	        // Check which specific status changed, prepare code, change state and write new status into the old one.
	        IF (#i_UDT_DimensionsCheckStatus.Specific.ParcelTooLongError <> #s_UDT_DimensionsCheckStatusOld.Specific.ParcelTooLongError AND NOT #sx_SendAllProcedure)
	            OR (#sx_SendAllProcedure AND #ii_ErrorNumber = 0)
	        THEN
	            #sdi_Code := "DB_MFC_ErrorCode".DimensionsCheck_v2.ParcelTooLongError;
	            #si_State := BOOL_TO_INT(#i_UDT_DimensionsCheckStatus.Specific.ParcelTooLongError);
	            #s_UDT_DimensionsCheckStatusOld.Specific.ParcelTooLongError := #i_UDT_DimensionsCheckStatus.Specific.ParcelTooLongError;
	            #sx_ItemErrorMessageReq := TRUE;
	            #ii_ErrorNumber += 1;
	        ELSIF (#i_UDT_DimensionsCheckStatus.Specific.ParcelTooShortError <> #s_UDT_DimensionsCheckStatusOld.Specific.ParcelTooShortError AND NOT #sx_SendAllProcedure)
	            OR (#sx_SendAllProcedure AND #ii_ErrorNumber = 1)
	        THEN
	            #sdi_Code := "DB_MFC_ErrorCode".DimensionsCheck_v2.ParcelTooShortError;
	            #si_State := BOOL_TO_INT(#i_UDT_DimensionsCheckStatus.Specific.ParcelTooShortError);
	            #s_UDT_DimensionsCheckStatusOld.Specific.ParcelTooShortError := #i_UDT_DimensionsCheckStatus.Specific.ParcelTooShortError;
	            #sx_ItemErrorMessageReq := TRUE;
	            #ii_ErrorNumber += 1;
	        ELSIF (#i_UDT_DimensionsCheckStatus.Specific.ParcelTooHighError <> #s_UDT_DimensionsCheckStatusOld.Specific.ParcelTooHighError AND NOT #sx_SendAllProcedure)
	            OR (#sx_SendAllProcedure AND #ii_ErrorNumber = 2)
	        THEN
	            #sdi_Code := "DB_MFC_ErrorCode".DimensionsCheck_v2.ParcelTooHighError;
	            #si_State := BOOL_TO_INT(#i_UDT_DimensionsCheckStatus.Specific.ParcelTooHighError);
	            #s_UDT_DimensionsCheckStatusOld.Specific.ParcelTooHighError := #i_UDT_DimensionsCheckStatus.Specific.ParcelTooHighError;
	            #sx_ItemErrorMessageReq := TRUE;
	            #ii_ErrorNumber += 1;
	        ELSIF (#i_UDT_DimensionsCheckStatus.Specific.ParcelTooLowError <> #s_UDT_DimensionsCheckStatusOld.Specific.ParcelTooLowError AND NOT #sx_SendAllProcedure)
	            OR (#sx_SendAllProcedure AND #ii_ErrorNumber = 3)
	        THEN
	            #sdi_Code := "DB_MFC_ErrorCode".DimensionsCheck_v2.ParcelTooLowError;
	            #si_State := BOOL_TO_INT(#i_UDT_DimensionsCheckStatus.Specific.ParcelTooLowError);
	            #s_UDT_DimensionsCheckStatusOld.Specific.ParcelTooLowError := #i_UDT_DimensionsCheckStatus.Specific.ParcelTooLowError;
	            #sx_ItemErrorMessageReq := TRUE;
	            #ii_ErrorNumber += 1;
	        ELSIF (#i_UDT_DimensionsCheckStatus.Specific.ParcelTooWideError <> #s_UDT_DimensionsCheckStatusOld.Specific.ParcelTooWideError AND NOT #sx_SendAllProcedure)
	            OR (#sx_SendAllProcedure AND #ii_ErrorNumber = 4)
	        THEN
	            #sdi_Code := "DB_MFC_ErrorCode".DimensionsCheck_v2.ParcelTooWideError;
	            #si_State := BOOL_TO_INT(#i_UDT_DimensionsCheckStatus.Specific.ParcelTooWideError);
	            #s_UDT_DimensionsCheckStatusOld.Specific.ParcelTooWideError := #i_UDT_DimensionsCheckStatus.Specific.ParcelTooWideError;
	            #sx_ItemErrorMessageReq := TRUE;
	            #ii_ErrorNumber += 1;
	        ELSIF (#i_UDT_DimensionsCheckStatus.Specific.ParcelTooNarrowError <> #s_UDT_DimensionsCheckStatusOld.Specific.ParcelTooNarrowError AND NOT #sx_SendAllProcedure)
	            OR (#sx_SendAllProcedure AND #ii_ErrorNumber = 5)
	        THEN
	            #sdi_Code := "DB_MFC_ErrorCode".DimensionsCheck_v2.ParcelTooNarrowError;
	            #si_State := BOOL_TO_INT(#i_UDT_DimensionsCheckStatus.Specific.ParcelTooNarrowError);
	            #s_UDT_DimensionsCheckStatusOld.Specific.ParcelTooNarrowError := #i_UDT_DimensionsCheckStatus.Specific.ParcelTooNarrowError;
	            #sx_ItemErrorMessageReq := TRUE;
	            #ii_ErrorNumber += 1;
	        ELSIF (#i_UDT_DimensionsCheckStatus.Specific.IncorrectParcelOrientationError <> #s_UDT_DimensionsCheckStatusOld.Specific.IncorrectParcelOrientationError AND NOT #sx_SendAllProcedure)
	            OR (#sx_SendAllProcedure AND #ii_ErrorNumber = 6)
	        THEN
	            #sdi_Code := "DB_MFC_ErrorCode".DimensionsCheck_v2.IncorrectParcelOrientationError;
	            #si_State := BOOL_TO_INT(#i_UDT_DimensionsCheckStatus.Specific.IncorrectParcelOrientationError);
	            #s_UDT_DimensionsCheckStatusOld.Specific.IncorrectParcelOrientationError := #i_UDT_DimensionsCheckStatus.Specific.IncorrectParcelOrientationError;
	            #sx_ItemErrorMessageReq := TRUE;
	            #ii_ErrorNumber += 1;
	        ELSIF (#i_UDT_DimensionsCheckStatus.Specific.GeneralError <> #s_UDT_DimensionsCheckStatusOld.Specific.GeneralError AND NOT #sx_SendAllProcedure)
	            OR (#sx_SendAllProcedure AND #ii_ErrorNumber = 7)
	        THEN
	            #sdi_Code := "DB_MFC_ErrorCode".DimensionsCheck_v2.GeneralError;
	            #si_State := BOOL_TO_INT(#i_UDT_DimensionsCheckStatus.Specific.GeneralError);
	            #s_UDT_DimensionsCheckStatusOld.Specific.GeneralError := #i_UDT_DimensionsCheckStatus.Specific.GeneralError;
	            #sx_ItemErrorMessageReq := TRUE;
	            #ii_ErrorNumber += 1;
	        ELSIF (#i_UDT_DimensionsCheckStatus.Specific.DisabledGeneralFunctionality <> #s_UDT_DimensionsCheckStatusOld.Specific.DisabledGeneralFunctionality AND NOT #sx_SendAllProcedure)
	            OR (#sx_SendAllProcedure AND #ii_ErrorNumber = 8)
	        THEN
	            #sdi_Code := "DB_MFC_ErrorCode".DimensionsCheck_v2.DisabledGeneralFunctionality;
	            #si_State := BOOL_TO_INT(#i_UDT_DimensionsCheckStatus.Specific.DisabledGeneralFunctionality);
	            #s_UDT_DimensionsCheckStatusOld.Specific.DisabledGeneralFunctionality := #i_UDT_DimensionsCheckStatus.Specific.DisabledGeneralFunctionality;
	            #sx_ItemErrorMessageReq := TRUE;
	            #ii_ErrorNumber += 1;
	        ELSIF (#i_UDT_DimensionsCheckStatus.Specific.DisabledTooLongParcel <> #s_UDT_DimensionsCheckStatusOld.Specific.DisabledTooLongParcel AND NOT #sx_SendAllProcedure)
	            OR (#sx_SendAllProcedure AND #ii_ErrorNumber = 9)
	        THEN
	            #sdi_Code := "DB_MFC_ErrorCode".DimensionsCheck_v2.DisabledTooLongParcel;
	            #si_State := BOOL_TO_INT(#i_UDT_DimensionsCheckStatus.Specific.DisabledTooLongParcel);
	            #s_UDT_DimensionsCheckStatusOld.Specific.DisabledTooLongParcel := #i_UDT_DimensionsCheckStatus.Specific.DisabledTooLongParcel;
	            #sx_ItemErrorMessageReq := TRUE;
	            #ii_ErrorNumber += 1;
	        ELSIF (#i_UDT_DimensionsCheckStatus.Specific.DisabledTooShortParcelError <> #s_UDT_DimensionsCheckStatusOld.Specific.DisabledTooShortParcelError AND NOT #sx_SendAllProcedure)
	            OR (#sx_SendAllProcedure AND #ii_ErrorNumber = 10)
	        THEN
	            #sdi_Code := "DB_MFC_ErrorCode".DimensionsCheck_v2.DisabledTooShortParcelError;
	            #si_State := BOOL_TO_INT(#i_UDT_DimensionsCheckStatus.Specific.DisabledTooShortParcelError);
	            #s_UDT_DimensionsCheckStatusOld.Specific.DisabledTooShortParcelError := #i_UDT_DimensionsCheckStatus.Specific.DisabledTooShortParcelError;
	            #sx_ItemErrorMessageReq := TRUE;
	            #ii_ErrorNumber += 1;
	        ELSIF (#i_UDT_DimensionsCheckStatus.Specific.DisabledTooHighParcelError <> #s_UDT_DimensionsCheckStatusOld.Specific.DisabledTooHighParcelError AND NOT #sx_SendAllProcedure)
	            OR (#sx_SendAllProcedure AND #ii_ErrorNumber = 11)
	        THEN
	            #sdi_Code := "DB_MFC_ErrorCode".DimensionsCheck_v2.DisabledTooHighParcelError;
	            #si_State := BOOL_TO_INT(#i_UDT_DimensionsCheckStatus.Specific.DisabledTooHighParcelError);
	            #s_UDT_DimensionsCheckStatusOld.Specific.DisabledTooHighParcelError := #i_UDT_DimensionsCheckStatus.Specific.DisabledTooHighParcelError;
	            #sx_ItemErrorMessageReq := TRUE;
	            #ii_ErrorNumber += 1;
	        ELSIF (#i_UDT_DimensionsCheckStatus.Specific.DisabledTooLowParcelError <> #s_UDT_DimensionsCheckStatusOld.Specific.DisabledTooLowParcelError AND NOT #sx_SendAllProcedure)
	            OR (#sx_SendAllProcedure AND #ii_ErrorNumber = 12)
	        THEN
	            #sdi_Code := "DB_MFC_ErrorCode".DimensionsCheck_v2.DisabledTooLowParcelError;
	            #si_State := BOOL_TO_INT(#i_UDT_DimensionsCheckStatus.Specific.DisabledTooLowParcelError);
	            #s_UDT_DimensionsCheckStatusOld.Specific.DisabledTooLowParcelError := #i_UDT_DimensionsCheckStatus.Specific.DisabledTooLowParcelError;
	            #sx_ItemErrorMessageReq := TRUE;
	            #ii_ErrorNumber += 1;
	        ELSIF (#i_UDT_DimensionsCheckStatus.Specific.DisabledTooWideParcelError <> #s_UDT_DimensionsCheckStatusOld.Specific.DisabledTooWideParcelError AND NOT #sx_SendAllProcedure)
	            OR (#sx_SendAllProcedure AND #ii_ErrorNumber = 13)
	        THEN
	            #sdi_Code := "DB_MFC_ErrorCode".DimensionsCheck_v2.DisabledTooWideParcelError;
	            #si_State := BOOL_TO_INT(#i_UDT_DimensionsCheckStatus.Specific.DisabledTooWideParcelError);
	            #s_UDT_DimensionsCheckStatusOld.Specific.DisabledTooWideParcelError := #i_UDT_DimensionsCheckStatus.Specific.DisabledTooWideParcelError;
	            #sx_ItemErrorMessageReq := TRUE;
	            #ii_ErrorNumber += 1;
	        ELSIF (#i_UDT_DimensionsCheckStatus.Specific.DisabledTooNarrowParcelError <> #s_UDT_DimensionsCheckStatusOld.Specific.DisabledTooNarrowParcelError AND NOT #sx_SendAllProcedure)
	            OR (#sx_SendAllProcedure AND #ii_ErrorNumber = 14)
	        THEN
	            #sdi_Code := "DB_MFC_ErrorCode".DimensionsCheck_v2.DisabledTooNarrowParcelError;
	            #si_State := BOOL_TO_INT(#i_UDT_DimensionsCheckStatus.Specific.DisabledTooNarrowParcelError);
	            #s_UDT_DimensionsCheckStatusOld.Specific.DisabledTooNarrowParcelError := #i_UDT_DimensionsCheckStatus.Specific.DisabledTooNarrowParcelError;
	            #sx_ItemErrorMessageReq := TRUE;
	            #ii_ErrorNumber += 1;
	        ELSIF (#i_UDT_DimensionsCheckStatus.Specific.DisabledParcelOrientationError <> #s_UDT_DimensionsCheckStatusOld.Specific.DisabledParcelOrientationError AND NOT #sx_SendAllProcedure)
	            OR (#sx_SendAllProcedure AND #ii_ErrorNumber = 15)
	        THEN
	            #sdi_Code := "DB_MFC_ErrorCode".DimensionsCheck_v2.DisabledParcelOrientationError;
	            #si_State := BOOL_TO_INT(#i_UDT_DimensionsCheckStatus.Specific.DisabledParcelOrientationError);
	            #s_UDT_DimensionsCheckStatusOld.Specific.DisabledParcelOrientationError := #i_UDT_DimensionsCheckStatus.Specific.DisabledParcelOrientationError;
	            #sx_ItemErrorMessageReq := TRUE;
	            #sx_SendAllProcedure := FALSE;
	            #ii_ErrorNumber += 1;
	        END_IF;
	    END_IF;
	END_REGION

	REGION 4 - Write message components to the item error structure

	    #s_UDT_ItemError.ItemNumber := #i_UDT_EquipmentNumber;
	    #s_UDT_ItemError.Error := #sdi_Code;
	    #s_UDT_ItemError.State := #si_State;
	    #s_UDT_ItemError.Masked := 1;

	END_REGION

	REGION 5 - Write message components to the item status structure

	    #s_UDT_ItemStatus.Group := #i_UDT_EquipmentNumber.Group;
	    #s_UDT_ItemStatus.Node := #i_UDT_EquipmentNumber.Node;
	    #s_UDT_ItemStatus.Status := #si_ItemStatus;

	END_REGION

	REGION 6 - Prepare messages to the MFC

	    // If item error message required signal is set, prepare the item error message.
	    IF (#sx_ItemErrorMessageReq)
	    THEN
	        #s_FB_ItemError(i_UDT_ItemErrorBody := #s_UDT_ItemError,
	                        ii_MessageGroup := 1,
	                        ix_FlagRetry := FALSE,
	                        idi_TimeSpan := 0,
	                        qx_Error => #sx_ItemErrorBlockError,
	                        qx_Warning => #sx_ItemErrorBlockWarning,
	                        iq_UDT_FifoHeader := #iq_UDT_FifoHeader,
	                        iqs_FifoData := #iqs_FifoData,
	                        iqdi_MessageSequenceNumber := #iqdi_MessageSequenceNumber);
	    END_IF;

	    // If item status message required signal is set, prepare the item error message.
	    IF (#sx_ItemStatusMessageReq)
	    THEN
	        #s_FB_ItemStatus(i_UDT_ItemStatusBody := #s_UDT_ItemStatus,
	                         ii_MessageGroup := 1,
	                         ix_FlagRetry := FALSE,
	                         idi_TimeSpan := 0,
	                         qx_Error => #sx_ItemStatusBlockError,
	                         qx_Warning => #sx_ItemStatusBlockWarning,
	                         iq_UDT_FifoHeader := #iq_UDT_FifoHeader,
	                         iqs_FifoData := #iqs_FifoData,
	                         iqdi_MessageSequenceNumber := #iqdi_MessageSequenceNumber);
	    END_IF;

	END_REGION

	REGION 7 - Write outputs

	    // Prepare collective output error.
	    #qx_Error :=
	    #sx_ItemErrorBlockError
	    OR #sx_ItemStatusBlockError
	    OR #sx_FIFOError;

	    // Prepare collective output warning.
	    #qx_Warning :=
	    #sx_ItemErrorBlockWarning
	    OR #sx_ItemStatusBlockWarning
	    OR #sx_FIFOWarning;

	END_REGION




END_FUNCTION_BLOCK

FUNCTION_BLOCK "FB_MFC_Visu_RetractableRoller_Status"
{ S7_Optimized_Access := 'TRUE' }
VERSION : 0.1
// ATTRIBUTES
// AUTO_NUMBER = True
// BLOCK_NUMBER = 157
// END_ATTRIBUTES
   VAR_INPUT
      i_UDT_RetractrableRollerStatus { ExternalAccessible := 'False'; ExternalVisible := 'False'; ExternalWritable := 'False'} : "UDT_RetractrableRoller_Status";   // RetractrableRoller status structure
      i_UDT_EquipmentNumber { ExternalAccessible := 'False'; ExternalVisible := 'False'; ExternalWritable := 'False'} : "UDT_EquipmentNumber";   // Item number
      ix_SendAllErrorsState { ExternalAccessible := 'False'; ExternalVisible := 'False'; ExternalWritable := 'False'} : Bool;   // True - update all the messages
      ix_MFCConnected { ExternalAccessible := 'False'; ExternalVisible := 'False'; ExternalWritable := 'False'} : Bool;   // True - A connection to the MFC has been established
      ix_CollectiveReset { ExternalAccessible := 'False'; ExternalVisible := 'False'; ExternalWritable := 'False'} : Bool;   // True - Collective reset command of all system controls
   END_VAR

   VAR_OUTPUT
      qx_Error { ExternalAccessible := 'False'; ExternalVisible := 'False'; ExternalWritable := 'False'} : Bool;   // Block error
      qx_Warning { ExternalAccessible := 'False'; ExternalVisible := 'False'; ExternalWritable := 'False'} : Bool;   // Block warning
   END_VAR

   VAR_IN_OUT
      iq_UDT_FifoHeader : "UDT_FifoHeader";   // FIFO header
      iqs_FifoData : Array[*] of "UDT_MessageV2";   // FIFO data buffer
      iqdi_MessageSequenceNumber { ExternalAccessible := 'False'; ExternalVisible := 'False'; ExternalWritable := 'False'} : DInt;   // Message number
   END_VAR

   VAR
      s_FB_ItemError { ExternalAccessible := 'False'; ExternalVisible := 'False'; ExternalWritable := 'False'; S7_SetPoint := 'False'} : "FB_ItemError";   // Item error block's instance
      s_FB_ItemStatus { ExternalAccessible := 'False'; ExternalVisible := 'False'; ExternalWritable := 'False'; S7_SetPoint := 'False'} : "FB_ItemStatus";   // Item status block's instance
      ss_FIFOStatus { ExternalAccessible := 'False'; ExternalVisible := 'False'; ExternalWritable := 'False'; S7_SetPoint := 'False'} : "UDT_FifoStatus";   // Status structure
      s_UDT_Message { ExternalAccessible := 'False'; ExternalVisible := 'False'; ExternalWritable := 'False'; S7_SetPoint := 'False'} : "UDT_MessageV2";   // Message
      s_UDT_RetractrableRollerOld { ExternalAccessible := 'False'; ExternalVisible := 'False'; ExternalWritable := 'False'; S7_SetPoint := 'False'} : "UDT_RetractrableRoller_Status";   // RetractrableRoller status structure
      s_UDT_ItemError { ExternalAccessible := 'False'; ExternalVisible := 'False'; ExternalWritable := 'False'; S7_SetPoint := 'False'} : "UDT_ItemError";   // Item error message body structure
      s_UDT_ItemStatus { ExternalAccessible := 'False'; ExternalVisible := 'False'; ExternalWritable := 'False'; S7_SetPoint := 'False'} : "UDT_ItemStatus";   // Item status message body structure
      s_R_TRIG_Connection {InstructionName := 'R_TRIG'; LibVersion := '1.0'; ExternalAccessible := 'False'; ExternalVisible := 'False'; ExternalWritable := 'False'; S7_SetPoint := 'False'} : R_TRIG;   // Rising edge trigger connection reastablished
      s_F_TRIG_SendAllErrors {InstructionName := 'F_TRIG'; LibVersion := '1.0'; ExternalAccessible := 'False'; ExternalVisible := 'False'; ExternalWritable := 'False'; S7_SetPoint := 'False'} : F_TRIG;   // Falling edge trigger from signal send all errors
      sdi_Code { ExternalAccessible := 'False'; ExternalVisible := 'False'; ExternalWritable := 'False'} : DInt;   // Error code
      si_ItemStatus { ExternalAccessible := 'False'; ExternalVisible := 'False'; ExternalWritable := 'False'} : Int;   // Item status
      ii_ErrorNumber { ExternalAccessible := 'False'; ExternalVisible := 'False'; ExternalWritable := 'False'} : Int;   // Counter Error Number
      si_State { ExternalAccessible := 'False'; ExternalVisible := 'False'; ExternalWritable := 'False'} : Int;   // Error state
      sx_ItemErrorMessageReq { ExternalAccessible := 'False'; ExternalVisible := 'False'; ExternalWritable := 'False'} : Bool;   // Item error message required
      sx_ItemStatusMessageReq { ExternalAccessible := 'False'; ExternalVisible := 'False'; ExternalWritable := 'False'} : Bool;   // Item status message required
      sx_SendAllProcedure { ExternalAccessible := 'False'; ExternalVisible := 'False'; ExternalWritable := 'False'} : Bool;   // Send all procedure
      sx_FIFOError { ExternalAccessible := 'False'; ExternalVisible := 'False'; ExternalWritable := 'False'} : Bool;   // FIFO error
      sx_FIFOWarning { ExternalAccessible := 'False'; ExternalVisible := 'False'; ExternalWritable := 'False'} : Bool;   // FIFO warning
      sx_ItemErrorBlockError { ExternalAccessible := 'False'; ExternalVisible := 'False'; ExternalWritable := 'False'} : Bool;   // Item error block error
      sx_ItemErrorBlockWarning { ExternalAccessible := 'False'; ExternalVisible := 'False'; ExternalWritable := 'False'} : Bool;   // Item error block warning
      sx_ItemStatusBlockError { ExternalAccessible := 'False'; ExternalVisible := 'False'; ExternalWritable := 'False'} : Bool;   // Item status block error
      sx_ItemStatusBlockWarning { ExternalAccessible := 'False'; ExternalVisible := 'False'; ExternalWritable := 'False'} : Bool;   // Item status block warning
   END_VAR


BEGIN
	(*
	----------------------------------------------------------------------------------------
	|                                                                                      |
	|  Copyright  2023             FORTNA Europe BV                                        |
	|  All Rights Reserved         Netherlands                                             |
	|                                                                                      |
	----------------------------------------------------------------------------------------
	Version history:
	Date        | Version   | Author       | Remark
	----------------------------------------------------------------------------------------
	09/05/2023  | 1.0       | M. Diebel   | Release TIA 17 | DHL Munich 2023
	13/03/2023  | 1.1       | S. Nieswiec | Updated for new Baseline
	*)


	REGION 1 - Initialize message required signals

	    #sx_ItemErrorMessageReq := FALSE;
	    #sx_ItemStatusMessageReq := FALSE;

	    // On connection reestablish send last remembered status and error state ( status only when it's diffrent then 0 )
	    #s_R_TRIG_Connection(CLK := #ix_MFCConnected);

	    IF #s_R_TRIG_Connection.Q AND #si_ItemStatus <> 0
	    THEN
	        #sx_ItemStatusMessageReq := TRUE;
	    END_IF;

	    IF #s_R_TRIG_Connection.Q
	    THEN
	        #sx_ItemErrorMessageReq := TRUE;
	    END_IF;

	    // Prepare trigger on the collective reset signal.
	    #s_F_TRIG_SendAllErrors(CLK := #ix_SendAllErrorsState);

	    // When collective reset will go down, start send every equipment errors.
	    IF #s_F_TRIG_SendAllErrors.Q AND NOT #sx_SendAllProcedure
	    THEN
	        #ii_ErrorNumber := 0;
	        #sx_SendAllProcedure := TRUE;
	    END_IF;

	END_REGION

	REGION 2 - FIFO header status update

	    // Mode 'S' - FIFO register status update.
	    "FC_Fifo"(ic_Mode := 'S',
	              qUDT_Status => #ss_FIFOStatus,
	              qx_Error => #sx_FIFOError,
	              qx_Warning => #sx_FIFOWarning,
	              iqv_Data := #s_UDT_Message,
	              iqUDT_FifoHeader := #iq_UDT_FifoHeader,
	              iqv_DataBuffer := #iqs_FifoData);

	END_REGION

	REGION 3 - Prepare message data

	    // When there is no reset errors command, update status and errors.
	    IF NOT #ix_CollectiveReset
	        AND NOT #ss_FIFOStatus.FifoPreFull
	    THEN
	        // Status
	        IF (#i_UDT_RetractrableRollerStatus.Status <> #s_UDT_RetractrableRollerOld.Status OR (#sx_SendAllProcedure AND #ii_ErrorNumber = 0))
	        THEN
	            #sx_ItemStatusMessageReq := TRUE;
	            #si_ItemStatus := #i_UDT_RetractrableRollerStatus.Status;
	            #s_UDT_RetractrableRollerOld.Status := #i_UDT_RetractrableRollerStatus.Status;
	        END_IF;


	        // Check which specific status changed, prepare code, change state and write new status into the old one.
	        IF (#i_UDT_RetractrableRollerStatus.Specific.NoHomePosition <> #s_UDT_RetractrableRollerOld.Specific.NoHomePosition AND NOT #sx_SendAllProcedure)
	            OR (#sx_SendAllProcedure AND #ii_ErrorNumber = 0)
	        THEN
	            #sdi_Code := "DB_MFC_ErrorCode".Retractable.NoHomePosition;
	            #si_State := BOOL_TO_INT(#i_UDT_RetractrableRollerStatus.Specific.NoHomePosition);
	            #s_UDT_RetractrableRollerOld.Specific.NoHomePosition := #i_UDT_RetractrableRollerStatus.Specific.NoHomePosition;
	            #sx_ItemErrorMessageReq := TRUE;
	            #ii_ErrorNumber += 1;
	        ELSIF (#i_UDT_RetractrableRollerStatus.Specific.RollerError <> #s_UDT_RetractrableRollerOld.Specific.RollerError AND NOT #sx_SendAllProcedure)
	            OR (#sx_SendAllProcedure AND #ii_ErrorNumber = 1)
	        THEN
	            #sdi_Code := "DB_MFC_ErrorCode".Retractable.Errorr;
	            #si_State := BOOL_TO_INT(#i_UDT_RetractrableRollerStatus.Specific.RollerError);
	            #s_UDT_RetractrableRollerOld.Specific.RollerError := #i_UDT_RetractrableRollerStatus.Specific.RollerError;
	            #sx_ItemErrorMessageReq := TRUE;
	            #sx_SendAllProcedure := FALSE;
	        END_IF;
	    END_IF;
	END_REGION

	REGION 4 - Write message components to the item error structure

	    #s_UDT_ItemError.ItemNumber := #i_UDT_EquipmentNumber;
	    #s_UDT_ItemError.Error := #sdi_Code;
	    #s_UDT_ItemError.State := #si_State;
	    #s_UDT_ItemError.Masked := 1;

	END_REGION

	REGION 5 - Write message components to the item status structure

	    #s_UDT_ItemStatus.Group := #i_UDT_EquipmentNumber.Group;
	    #s_UDT_ItemStatus.Node := #i_UDT_EquipmentNumber.Node;
	    #s_UDT_ItemStatus.Status := #si_ItemStatus;

	END_REGION

	REGION 6 - Prepare messages to the MFC

	    // If item error message required signal is set, prepare the item error message.
	    IF (#sx_ItemErrorMessageReq)
	    THEN
	        #s_FB_ItemError(i_UDT_ItemErrorBody := #s_UDT_ItemError,
	                        ii_MessageGroup := 1,
	                        ix_FlagRetry := FALSE,
	                        idi_TimeSpan := 0,
	                        qx_Error => #sx_ItemErrorBlockError,
	                        qx_Warning => #sx_ItemErrorBlockWarning,
	                        iq_UDT_FifoHeader := #iq_UDT_FifoHeader,
	                        iqs_FifoData := #iqs_FifoData,
	                        iqdi_MessageSequenceNumber := #iqdi_MessageSequenceNumber);
	    END_IF;

	    // If item status message required signal is set, prepare the item error message.
	    IF (#sx_ItemStatusMessageReq)
	    THEN
	        #s_FB_ItemStatus(i_UDT_ItemStatusBody := #s_UDT_ItemStatus,
	                         ii_MessageGroup := 1,
	                         ix_FlagRetry := FALSE,
	                         idi_TimeSpan := 0,
	                         qx_Error => #sx_ItemStatusBlockError,
	                         qx_Warning => #sx_ItemStatusBlockWarning,
	                         iq_UDT_FifoHeader := #iq_UDT_FifoHeader,
	                         iqs_FifoData := #iqs_FifoData,
	                         iqdi_MessageSequenceNumber := #iqdi_MessageSequenceNumber);
	    END_IF;

	END_REGION

	REGION 7 - Write outputs

	    // Prepare collective output error.
	    #qx_Error :=
	    #sx_ItemErrorBlockError
	    OR #sx_ItemStatusBlockError
	    OR #sx_FIFOError;

	    // Prepare collective output warning.
	    #qx_Warning :=
	    #sx_ItemErrorBlockWarning
	    OR #sx_ItemStatusBlockWarning
	    OR #sx_FIFOWarning;

	END_REGION


END_FUNCTION_BLOCK

FUNCTION_BLOCK "FB_MFC_Visu_RIO_Status"
{ S7_Optimized_Access := 'TRUE' }
VERSION : 0.1
// ATTRIBUTES
// AUTO_NUMBER = True
// BLOCK_NUMBER = 158
// END_ATTRIBUTES
   VAR_INPUT
      i_UDT_RIOStatus { ExternalAccessible := 'False'; ExternalVisible := 'False'; ExternalWritable := 'False'} : "UDT_RIOStatus";   // RIO status structure
      i_UDT_EquipmentNumber { ExternalAccessible := 'False'; ExternalVisible := 'False'; ExternalWritable := 'False'} : "UDT_EquipmentNumber";   // Item number
      ix_SendAllErrorsState { ExternalAccessible := 'False'; ExternalVisible := 'False'; ExternalWritable := 'False'} : Bool;   // True - update all the messages
      ix_MFCConnected { ExternalAccessible := 'False'; ExternalVisible := 'False'; ExternalWritable := 'False'} : Bool;   // True - A connection to the MFC has been established
      ix_CollectiveReset { ExternalAccessible := 'False'; ExternalVisible := 'False'; ExternalWritable := 'False'} : Bool;   // True - Collective reset command of all system controls
   END_VAR

   VAR_OUTPUT
      qx_Error { ExternalAccessible := 'False'; ExternalVisible := 'False'; ExternalWritable := 'False'} : Bool;   // Block error
      qx_Warning { ExternalAccessible := 'False'; ExternalVisible := 'False'; ExternalWritable := 'False'} : Bool;   // Block warning
   END_VAR

   VAR_IN_OUT
      iq_UDT_FifoHeader : "UDT_FifoHeader";   // FIFO header
      iqs_FifoData : Array[*] of "UDT_MessageV2";   // FIFO data buffer
      iqdi_MessageSequenceNumber { ExternalAccessible := 'False'; ExternalVisible := 'False'; ExternalWritable := 'False'} : DInt;   // Message number
   END_VAR

   VAR
      s_FB_ItemStatus { ExternalAccessible := 'False'; ExternalVisible := 'False'; ExternalWritable := 'False'; S7_SetPoint := 'False'} : "FB_ItemStatus";   // Item status block's instance
      s_FB_ItemError { ExternalAccessible := 'False'; ExternalVisible := 'False'; ExternalWritable := 'False'; S7_SetPoint := 'False'} : "FB_ItemError";   // Item error block's instance
      ss_FIFOStatus { ExternalAccessible := 'False'; ExternalVisible := 'False'; ExternalWritable := 'False'; S7_SetPoint := 'False'} : "UDT_FifoStatus";   // Status structure
      s_UDT_Message { ExternalAccessible := 'False'; ExternalVisible := 'False'; ExternalWritable := 'False'; S7_SetPoint := 'False'} : "UDT_MessageV2";   // Message
      s_UDT_RIOOld { ExternalAccessible := 'False'; ExternalVisible := 'False'; ExternalWritable := 'False'; S7_SetPoint := 'False'} : "UDT_RIOStatus";   // RIO old status structure
      s_UDT_ItemError { ExternalAccessible := 'False'; ExternalVisible := 'False'; ExternalWritable := 'False'; S7_SetPoint := 'False'} : "UDT_ItemError";   // Item error message body structure
      s_UDT_ItemStatus { ExternalAccessible := 'False'; ExternalVisible := 'False'; ExternalWritable := 'False'; S7_SetPoint := 'False'} : "UDT_ItemStatus";   // Item status message body structure
      s_F_TRIG_SendAllErrors {InstructionName := 'F_TRIG'; LibVersion := '1.0'; ExternalAccessible := 'False'; ExternalVisible := 'False'; ExternalWritable := 'False'; S7_SetPoint := 'False'} : F_TRIG;   // Falling edge trigger from signal send all errors
      s_R_TRIG_Connection {InstructionName := 'R_TRIG'; LibVersion := '1.0'; ExternalAccessible := 'False'; ExternalVisible := 'False'; ExternalWritable := 'False'; S7_SetPoint := 'False'} : R_TRIG;   // Rising edge trigger connection reastablished
      sdi_Code { ExternalAccessible := 'False'; ExternalVisible := 'False'; ExternalWritable := 'False'} : DInt;   // Error code
      si_ET { ExternalAccessible := 'False'; ExternalVisible := 'False'; ExternalWritable := 'False'} : Int;   // Value
      si_ItemStatus { ExternalAccessible := 'False'; ExternalVisible := 'False'; ExternalWritable := 'False'} : Int;   // Item status
      ii_ErrorNumber { ExternalAccessible := 'False'; ExternalVisible := 'False'; ExternalWritable := 'False'} : Int;   // Counter Error Number
      si_State { ExternalAccessible := 'False'; ExternalVisible := 'False'; ExternalWritable := 'False'} : Int;   // Error state
      sx_ItemErrorMessageReq { ExternalAccessible := 'False'; ExternalVisible := 'False'; ExternalWritable := 'False'} : Bool;   // Item error message required
      sx_ItemStatusMessageReq { ExternalAccessible := 'False'; ExternalVisible := 'False'; ExternalWritable := 'False'} : Bool;   // Item status message required
      sx_SendAllProcedure { ExternalAccessible := 'False'; ExternalVisible := 'False'; ExternalWritable := 'False'} : Bool;   // Send all procedure
      sx_FIFOError { ExternalAccessible := 'False'; ExternalVisible := 'False'; ExternalWritable := 'False'} : Bool;   // FIFO error
      sx_FIFOWarning { ExternalAccessible := 'False'; ExternalVisible := 'False'; ExternalWritable := 'False'} : Bool;   // FIFO warning
      sx_ItemErrorBlockError { ExternalAccessible := 'False'; ExternalVisible := 'False'; ExternalWritable := 'False'} : Bool;   // Item error block error
      sx_ItemErrorBlockWarning { ExternalAccessible := 'False'; ExternalVisible := 'False'; ExternalWritable := 'False'} : Bool;   // Item error block warning
      sx_ItemStatusBlockError { ExternalAccessible := 'False'; ExternalVisible := 'False'; ExternalWritable := 'False'} : Bool;   // Item status block error
      sx_ItemStatusBlockWarning { ExternalAccessible := 'False'; ExternalVisible := 'False'; ExternalWritable := 'False'} : Bool;   // Item status block warning
   END_VAR


BEGIN
	(*
	----------------------------------------------------------------------------------------
	|                                                                                      |
	|  Copyright  2023             FORTNA Europe BV                                        |
	|  All Rights Reserved         Netherlands                                             |
	|                                                                                      |
	----------------------------------------------------------------------------------------
	Version history:
	Date        | Version   | Author       | Remark
	----------------------------------------------------------------------------------------
	21/03/2023  | 1.0       | M. Diebel   | Release TIA 17 | DHL Munich 2023
	13/03/2023  | 1.1       | S. Nieswiec | Updated for new Baseline
	*)


	REGION 1 - Initialize message required signals

	    #sx_ItemErrorMessageReq := FALSE;
	    #sx_ItemStatusMessageReq := FALSE;

	    // On connection reestablish send last remembered status and error state ( status only when it's diffrent then 0 )
	    #s_R_TRIG_Connection(CLK := #ix_MFCConnected);

	    IF #s_R_TRIG_Connection.Q AND #si_ItemStatus <> 0
	    THEN
	        #sx_ItemStatusMessageReq := TRUE;
	    END_IF;

	    IF #s_R_TRIG_Connection.Q
	    THEN
	        #sx_ItemErrorMessageReq := TRUE;
	    END_IF;

	    // Prepare trigger on the collective reset signal.
	    #s_F_TRIG_SendAllErrors(CLK := #ix_SendAllErrorsState);

	    // When collective reset will go down, start send every equipment errors.
	    IF #s_F_TRIG_SendAllErrors.Q AND NOT #sx_SendAllProcedure
	    THEN
	        #ii_ErrorNumber := 0;
	        #sx_SendAllProcedure := TRUE;
	    END_IF;

	END_REGION

	REGION 2 - FIFO header status update

	    // Mode 'S' - FIFO register status update.
	    "FC_Fifo"(ic_Mode := 'S',
	              qUDT_Status => #ss_FIFOStatus,
	              qx_Error => #sx_FIFOError,
	              qx_Warning => #sx_FIFOWarning,
	              iqv_Data := #s_UDT_Message,
	              iqUDT_FifoHeader := #iq_UDT_FifoHeader,
	              iqv_DataBuffer := #iqs_FifoData);

	END_REGION

	REGION 3 - Prepare message data

	    // When there is no reset errors command, update status and errors.
	    IF NOT #ix_CollectiveReset
	        AND NOT #ss_FIFOStatus.FifoPreFull
	    THEN
	        // Status
	        IF (#i_UDT_RIOStatus.Status <> #s_UDT_RIOOld.Status OR (#sx_SendAllProcedure AND #ii_ErrorNumber = 0))
	        THEN
	            #sx_ItemStatusMessageReq := TRUE;
	            #si_ItemStatus := #i_UDT_RIOStatus.Status;
	            #s_UDT_RIOOld.Status := #i_UDT_RIOStatus.Status;
	        END_IF;


	        // Check which specific status changed, prepare code, change state and write new status into the old one.
	        IF (#i_UDT_RIOStatus.Specific.PNSlaveNotOnline <> #s_UDT_RIOOld.Specific.PNSlaveNotOnline AND NOT #sx_SendAllProcedure)
	            OR (#sx_SendAllProcedure AND #ii_ErrorNumber = 0)
	        THEN
	            #sdi_Code := "DB_MFC_ErrorCode".RIO.PNSlaveNotOnline;
	            #si_State := BOOL_TO_INT(#i_UDT_RIOStatus.Specific.PNSlaveNotOnline);
	            #s_UDT_RIOOld.Specific.PNSlaveNotOnline := #i_UDT_RIOStatus.Specific.PNSlaveNotOnline;
	            #sx_ItemErrorMessageReq := TRUE;
	            #ii_ErrorNumber += 1;
	        ELSIF (#i_UDT_RIOStatus.Specific.PNSlaveError <> #s_UDT_RIOOld.Specific.PNSlaveError AND NOT #sx_SendAllProcedure)
	            OR (#sx_SendAllProcedure AND #ii_ErrorNumber = 1)
	        THEN
	            #sdi_Code := "DB_MFC_ErrorCode".RIO.PNSlaveError;
	            #si_State := BOOL_TO_INT(#i_UDT_RIOStatus.Specific.PNSlaveError);
	            #s_UDT_RIOOld.Specific.PNSlaveError := #i_UDT_RIOStatus.Specific.PNSlaveError;
	            #sx_ItemErrorMessageReq := TRUE;
	            #ii_ErrorNumber += 1;
	        ELSIF (#i_UDT_RIOStatus.Specific.PNSlaveWarning <> #s_UDT_RIOOld.Specific.PNSlaveWarning AND NOT #sx_SendAllProcedure)
	            OR (#sx_SendAllProcedure AND #ii_ErrorNumber = 2)
	        THEN
	            #sdi_Code := "DB_MFC_ErrorCode".RIO.PNSlaveWarning;
	            #si_State := BOOL_TO_INT(#i_UDT_RIOStatus.Specific.PNSlaveWarning);
	            #s_UDT_RIOOld.Specific.PNSlaveWarning := #i_UDT_RIOStatus.Specific.PNSlaveWarning;
	            #sx_ItemErrorMessageReq := TRUE;
	            #sx_SendAllProcedure := FALSE;
	            #ii_ErrorNumber += 1;
	        ELSE

	            FOR #si_ET := 0 TO 31 DO

	                IF (#i_UDT_RIOStatus.Specific.ET200sp_ErrorModule[#si_ET] <> #s_UDT_RIOOld.Specific.ET200sp_ErrorModule[#si_ET])
	                THEN
	                    #sdi_Code := "DB_MFC_ErrorCode".RIO.ET200sp_ErrorModule[#si_ET];
	                    #si_State := BOOL_TO_INT(#i_UDT_RIOStatus.Specific.ET200sp_ErrorModule[#si_ET]);
	                    #s_UDT_RIOOld.Specific.ET200sp_ErrorModule[#si_ET] := #i_UDT_RIOStatus.Specific.ET200sp_ErrorModule[#si_ET];
	                    #sx_ItemErrorMessageReq := TRUE;
	                    EXIT;
	                END_IF;
	            END_FOR;
	        END_IF;

	    END_IF;
	END_REGION

	REGION 4 - Write message components to the item error structure

	    #s_UDT_ItemError.ItemNumber := #i_UDT_EquipmentNumber;
	    #s_UDT_ItemError.Error := #sdi_Code;
	    #s_UDT_ItemError.State := #si_State;
	    #s_UDT_ItemError.Masked := 1;

	END_REGION

	REGION 5 - Write message components to the item status structure

	    #s_UDT_ItemStatus.Group := #i_UDT_EquipmentNumber.Group;
	    #s_UDT_ItemStatus.Node := #i_UDT_EquipmentNumber.Node;
	    #s_UDT_ItemStatus.Status := #si_ItemStatus;

	END_REGION

	REGION 6 - Prepare messages to the MFC

	    // If item error message required signal is set, prepare the item error message.
	    IF (#sx_ItemErrorMessageReq)
	    THEN
	        #s_FB_ItemError(i_UDT_ItemErrorBody := #s_UDT_ItemError,
	                        ii_MessageGroup := 1,
	                        ix_FlagRetry := FALSE,
	                        idi_TimeSpan := 0,
	                        qx_Error => #sx_ItemErrorBlockError,
	                        qx_Warning => #sx_ItemErrorBlockWarning,
	                        iq_UDT_FifoHeader := #iq_UDT_FifoHeader,
	                        iqs_FifoData := #iqs_FifoData,
	                        iqdi_MessageSequenceNumber := #iqdi_MessageSequenceNumber);
	    END_IF;

	    // If item status message required signal is set, prepare the item error message.
	    IF (#sx_ItemStatusMessageReq)
	    THEN
	        #s_FB_ItemStatus(i_UDT_ItemStatusBody := #s_UDT_ItemStatus,
	                         ii_MessageGroup := 1,
	                         ix_FlagRetry := FALSE,
	                         idi_TimeSpan := 0,
	                         qx_Error => #sx_ItemStatusBlockError,
	                         qx_Warning => #sx_ItemStatusBlockWarning,
	                         iq_UDT_FifoHeader := #iq_UDT_FifoHeader,
	                         iqs_FifoData := #iqs_FifoData,
	                         iqdi_MessageSequenceNumber := #iqdi_MessageSequenceNumber);
	    END_IF;

	END_REGION

	REGION 7 - Write outputs

	    // Prepare collective output error.
	    #qx_Error :=
	    #sx_ItemErrorBlockError
	    OR #sx_ItemStatusBlockError
	    OR #sx_FIFOError;

	    // Prepare collective output warning.
	    #qx_Warning :=
	    #sx_ItemErrorBlockWarning
	    OR #sx_ItemStatusBlockWarning
	    OR #sx_FIFOWarning;

	END_REGION
END_FUNCTION_BLOCK

FUNCTION_BLOCK "FB_MFC_Visu_SystemControl_Status"
{ S7_Optimized_Access := 'TRUE' }
VERSION : 0.1
// ATTRIBUTES
// AUTO_NUMBER = True
// BLOCK_NUMBER = 159
// END_ATTRIBUTES
   VAR_INPUT
      i_UDT_SystemControlStatus { ExternalAccessible := 'False'; ExternalVisible := 'False'; ExternalWritable := 'False'} : "UDT_SystemControlStatus";   // System control status structure
      i_UDT_EquipmentNumber { ExternalAccessible := 'False'; ExternalVisible := 'False'; ExternalWritable := 'False'} : "UDT_EquipmentNumber";   // Item number
      ix_SendAllErrorsState { ExternalAccessible := 'False'; ExternalVisible := 'False'; ExternalWritable := 'False'} : Bool;   // True - update all the messages
      ix_MFCConnected { ExternalAccessible := 'False'; ExternalVisible := 'False'; ExternalWritable := 'False'} : Bool;   // True - A connection to the MFC has been established
      ix_CollectiveReset { ExternalAccessible := 'False'; ExternalVisible := 'False'; ExternalWritable := 'False'} : Bool;   // True - Collective reset command of all system controls
   END_VAR

   VAR_OUTPUT
      qx_Error { ExternalAccessible := 'False'; ExternalVisible := 'False'; ExternalWritable := 'False'} : Bool;   // Block error
      qx_Warning { ExternalAccessible := 'False'; ExternalVisible := 'False'; ExternalWritable := 'False'} : Bool;   // Block warning
   END_VAR

   VAR_IN_OUT
      iq_UDT_FifoHeader : "UDT_FifoHeader";   // FIFO header
      iqs_FifoData : Array[*] of "UDT_MessageV2";   // FIFO data buffer
      iqdi_MessageSequenceNumber { ExternalAccessible := 'False'; ExternalVisible := 'False'; ExternalWritable := 'False'} : DInt;   // Message number
   END_VAR

   VAR
      s_FB_ItemStatus { ExternalAccessible := 'False'; ExternalVisible := 'False'; ExternalWritable := 'False'; S7_SetPoint := 'False'} : "FB_ItemStatus";   // Item status block's instance
      s_FB_ItemError { ExternalAccessible := 'False'; ExternalVisible := 'False'; ExternalWritable := 'False'; S7_SetPoint := 'False'} : "FB_ItemError";   // Item error block's instance
      ss_FIFOStatus { ExternalAccessible := 'False'; ExternalVisible := 'False'; ExternalWritable := 'False'; S7_SetPoint := 'False'} : "UDT_FifoStatus";   // Status structure
      s_UDT_Message { ExternalAccessible := 'False'; ExternalVisible := 'False'; ExternalWritable := 'False'; S7_SetPoint := 'False'} : "UDT_MessageV2";   // Message
      s_UDT_SystemControlStatusOld { ExternalAccessible := 'False'; ExternalVisible := 'False'; ExternalWritable := 'False'; S7_SetPoint := 'False'} : "UDT_SystemControlStatus";   // System control old status structure
      s_UDT_ItemError { ExternalAccessible := 'False'; ExternalVisible := 'False'; ExternalWritable := 'False'; S7_SetPoint := 'False'} : "UDT_ItemError";   // Item error message body structure
      s_UDT_ItemStatus { ExternalAccessible := 'False'; ExternalVisible := 'False'; ExternalWritable := 'False'; S7_SetPoint := 'False'} : "UDT_ItemStatus";   // Item status message body structure
      s_F_TRIG_SendAllErrors {InstructionName := 'F_TRIG'; LibVersion := '1.0'; ExternalAccessible := 'False'; ExternalVisible := 'False'; ExternalWritable := 'False'; S7_SetPoint := 'False'} : F_TRIG;   // Falling edge trigger from signal send all errors
      s_R_TRIG_Connection {InstructionName := 'R_TRIG'; LibVersion := '1.0'; ExternalAccessible := 'False'; ExternalVisible := 'False'; ExternalWritable := 'False'; S7_SetPoint := 'False'} : R_TRIG;   // Rising edge trigger connection reastablished
      sdi_Code { ExternalAccessible := 'False'; ExternalVisible := 'False'; ExternalWritable := 'False'} : DInt;   // Error code
      si_ItemStatus { ExternalAccessible := 'False'; ExternalVisible := 'False'; ExternalWritable := 'False'} : Int;   // Item status
      ii_ErrorNumber { ExternalAccessible := 'False'; ExternalVisible := 'False'; ExternalWritable := 'False'} : Int;   // Counter Error Number
      si_State { ExternalAccessible := 'False'; ExternalVisible := 'False'; ExternalWritable := 'False'} : Int;   // Error state
      sx_ItemErrorMessageReq { ExternalAccessible := 'False'; ExternalVisible := 'False'; ExternalWritable := 'False'} : Bool;   // Item error message required
      sx_ItemStatusMessageReq { ExternalAccessible := 'False'; ExternalVisible := 'False'; ExternalWritable := 'False'} : Bool;   // Item status message required
      sx_SendAllProcedure { ExternalAccessible := 'False'; ExternalVisible := 'False'; ExternalWritable := 'False'} : Bool;   // Send all procedure
      sx_FIFOError { ExternalAccessible := 'False'; ExternalVisible := 'False'; ExternalWritable := 'False'} : Bool;   // FIFO error
      sx_FIFOWarning { ExternalAccessible := 'False'; ExternalVisible := 'False'; ExternalWritable := 'False'} : Bool;   // FIFO warning
      sx_ItemStatusBlockError { ExternalAccessible := 'False'; ExternalVisible := 'False'; ExternalWritable := 'False'} : Bool;   // Item status block error
      sx_ItemStatusBlockWarning { ExternalAccessible := 'False'; ExternalVisible := 'False'; ExternalWritable := 'False'} : Bool;   // Item status block warning
   END_VAR


BEGIN
	(*
	----------------------------------------------------------------------------------------
	|                                                                                      |
	|  Copyright  2023             FORTNA Europe BV                                        |
	|  All Rights Reserved         Netherlands                                             |
	|                                                                                      |
	----------------------------------------------------------------------------------------
	Version history:
	Date        | Version   | Author       | Remark
	----------------------------------------------------------------------------------------
	24/03/2023  | 1.0       | M. Diebel   | Release TIA 17 | DHL Munich 2023
	13/03/2023  | 1.1       | S. Nieswiec  | Updated for new Baseline
	*)


	REGION 1 - Initialize message required signals


	    #sx_ItemStatusMessageReq := FALSE;

	    // On connection reestablish send last remembered status and error state ( status only when it's diffrent then 0 )
	    #s_R_TRIG_Connection(CLK := #ix_MFCConnected);

	    IF #s_R_TRIG_Connection.Q AND #si_ItemStatus <> 0
	    THEN
	        #sx_ItemStatusMessageReq := TRUE;
	    END_IF;


	    // Prepare trigger on the collective reset signal.
	    #s_F_TRIG_SendAllErrors(CLK := #ix_SendAllErrorsState);

	    // When collective reset will go down, start send every equipment errors.
	    IF #s_F_TRIG_SendAllErrors.Q AND NOT #sx_SendAllProcedure
	    THEN
	        #ii_ErrorNumber := 0;
	        #sx_SendAllProcedure := TRUE;
	    END_IF;

	END_REGION


	REGION 2 - FIFO header status update

	    // Mode 'S' - FIFO register status update.
	    "FC_Fifo"(ic_Mode := 'S',
	              qUDT_Status => #ss_FIFOStatus,
	              qx_Error => #sx_FIFOError,
	              qx_Warning => #sx_FIFOWarning,
	              iqv_Data := #s_UDT_Message,
	              iqUDT_FifoHeader := #iq_UDT_FifoHeader,
	              iqv_DataBuffer := #iqs_FifoData);

	END_REGION


	REGION 3 - Prepare message data

	    // When there is no reset errors command, update status and errors.
	    IF NOT #ix_CollectiveReset
	        AND NOT #ss_FIFOStatus.FifoPreFull
	    THEN
	        // Status
	        IF (#i_UDT_SystemControlStatus.Status <> #s_UDT_SystemControlStatusOld.Status OR (#sx_SendAllProcedure AND #ii_ErrorNumber = 0))
	        THEN
	            #sx_ItemStatusMessageReq := TRUE;
	            #si_ItemStatus := #i_UDT_SystemControlStatus.Status;
	            #s_UDT_SystemControlStatusOld.Status := #i_UDT_SystemControlStatus.Status;
	            #sx_SendAllProcedure := FALSE;
	        END_IF;
	    END_IF;
	END_REGION


	REGION 4 - Write message components to the item status structure

	    #s_UDT_ItemStatus.Group := #i_UDT_EquipmentNumber.Group;
	    #s_UDT_ItemStatus.Node := #i_UDT_EquipmentNumber.Node;
	    #s_UDT_ItemStatus.Status := #si_ItemStatus;

	END_REGION

	REGION 5 - Prepare messages to the MFC

	    // If item status message required signal is set, prepare the item error message.
	    IF (#sx_ItemStatusMessageReq)
	    THEN
	        #s_FB_ItemStatus(i_UDT_ItemStatusBody := #s_UDT_ItemStatus,
	                         ii_MessageGroup := 1,
	                         ix_FlagRetry := FALSE,
	                         idi_TimeSpan := 0,
	                         qx_Error => #sx_ItemStatusBlockError,
	                         qx_Warning => #sx_ItemStatusBlockWarning,
	                         iq_UDT_FifoHeader := #iq_UDT_FifoHeader,
	                         iqs_FifoData := #iqs_FifoData,
	                         iqdi_MessageSequenceNumber := #iqdi_MessageSequenceNumber);
	    END_IF;

	END_REGION

	REGION 6 - Write outputs

	    // Prepare collective output error.
	    #qx_Error :=
	    #sx_ItemStatusBlockError
	    OR #sx_FIFOError;

	    // Prepare collective output warning.
	    #qx_Warning :=
	    #sx_ItemStatusBlockWarning
	    OR #sx_FIFOWarning;

	END_REGION
END_FUNCTION_BLOCK

FUNCTION_BLOCK "FB_MFC_Visu_Decode"
{ S7_Optimized_Access := 'TRUE' }
VERSION : 0.1
// ATTRIBUTES
// AUTO_NUMBER = True
// BLOCK_NUMBER = 143
// END_ATTRIBUTES
   VAR_INPUT
      iudi_HeartbeatTimeout { ExternalAccessible := 'False'; ExternalVisible := 'False'; ExternalWritable := 'False'} : UDInt;   //   Heartbeat timeout [ms]
      ix_Connected { ExternalAccessible := 'False'; ExternalVisible := 'False'; ExternalWritable := 'False'} : Bool;   //   TRUE when HB monitoring enable
      ix_ResetData { ExternalAccessible := 'False'; ExternalVisible := 'False'; ExternalWritable := 'False'} : Bool;   //   TRUE when reset statistics required
   END_VAR

   VAR_OUTPUT
      qx_Error { ExternalAccessible := 'False'; ExternalVisible := 'False'; ExternalWritable := 'False'} : Bool;   //   TRUE when collective block error occurred
      qx_Warning { ExternalAccessible := 'False'; ExternalVisible := 'False'; ExternalWritable := 'False'} : Bool;   //   TRUE when collective block warningoccurred
      qx_SendAllErrorsState { ExternalAccessible := 'False'; ExternalVisible := 'False'; ExternalWritable := 'False'} : Bool;
   END_VAR

   VAR_IN_OUT
      iqx_Reconnect { ExternalAccessible := 'False'; ExternalVisible := 'False'; ExternalWritable := 'False'} : Bool;   //   Reconnect connection
      iq_UDT_Statistics : "UDT_DecodeStatistics";   //   Decode statistics
      iq_UDT_FifoReceiveHeader : "UDT_FifoHeader";   //   FIFO receive header
      iqs_FifoReceiveData : Array[*] of "UDT_MessageV2";   //   FIFO receive data
   END_VAR

   VAR
      s_FB_TimerHeartbeatCheck { ExternalAccessible := 'False'; ExternalVisible := 'False'; ExternalWritable := 'False'; S7_SetPoint := 'False'} : "FB_TimerOnOffDelay";   //   MHS "FB_TimerOnOffDelay" - to measure the time of missing HB
      s_UDT_FifoMessage { ExternalAccessible := 'False'; ExternalVisible := 'False'; ExternalWritable := 'False'; S7_SetPoint := 'False'} : "UDT_MessageV2";   //   Buffer for fifos message
      s_UDT_MessageHeader { ExternalAccessible := 'False'; ExternalVisible := 'False'; ExternalWritable := 'False'; S7_SetPoint := 'False'} : "UDT_MessageHeaderV2";   //   Message header
      s_UDT_Heartbeat { ExternalAccessible := 'False'; ExternalVisible := 'False'; ExternalWritable := 'False'; S7_SetPoint := 'False'} : "UDT_MessageHeaderV2";   //   Heartbeat message
      s_UDT_SetDateTime { ExternalAccessible := 'False'; ExternalVisible := 'False'; ExternalWritable := 'False'; S7_SetPoint := 'False'} : "UDT_SetDateTimeBody";   //   Set date time message body
      s_UDT_MFCCommand { ExternalAccessible := 'False'; ExternalVisible := 'False'; ExternalWritable := 'False'; S7_SetPoint := 'False'} : "UDT_MFCCommandBody";   // MFC command message body
      s_R_TRIG_Connected {InstructionName := 'R_TRIG'; LibVersion := '1.0'; ExternalAccessible := 'False'; ExternalVisible := 'False'; ExternalWritable := 'False'; S7_SetPoint := 'False'} : R_TRIG;   //   Siemens "R_TRIG" - to prepare the rising edge trigger on "ix_Connected" signal
      s_R_TRIG_FirstConnection {InstructionName := 'R_TRIG'; LibVersion := '1.0'; ExternalAccessible := 'False'; ExternalVisible := 'False'; ExternalWritable := 'False'; S7_SetPoint := 'False'} : R_TRIG;
      s_F_TRIG_HeartbeatNotOk {InstructionName := 'F_TRIG'; LibVersion := '1.0'; ExternalAccessible := 'False'; ExternalVisible := 'False'; ExternalWritable := 'False'; S7_SetPoint := 'False'} : F_TRIG;   //   Siemens "F_TRIG" - to prepare the falling edge trigger on "sx_HeartbeatOk" signal
      ss_Status { ExternalAccessible := 'False'; ExternalVisible := 'False'; ExternalWritable := 'False'} : Struct   //   Status structure
         BadMessage { ExternalAccessible := 'False'; ExternalVisible := 'False'; ExternalWritable := 'False'} : Array[1..10] of "UDT_MessageV2";   //     Unknown message read
         FIFOReceiveStatus { ExternalAccessible := 'False'; ExternalVisible := 'False'; ExternalWritable := 'False'} : "UDT_FifoStatus";   //     Receive FIFO status structure
         FIFOReceiveError { ExternalAccessible := 'False'; ExternalVisible := 'False'; ExternalWritable := 'False'; S7_SetPoint := 'True'} : Bool;   //     FIFO error
         FIFOReceiveWarning { ExternalAccessible := 'False'; ExternalVisible := 'False'; ExternalWritable := 'False'} : Bool;   //     FIFO warning
         OperationModeError { ExternalAccessible := 'False'; ExternalVisible := 'False'; ExternalWritable := 'False'} : Bool;   //     Operation mode error
         OperationModeWarning { ExternalAccessible := 'False'; ExternalVisible := 'False'; ExternalWritable := 'False'} : Bool;   //     Operation mode warning
         OverflowModeError { ExternalAccessible := 'False'; ExternalVisible := 'False'; ExternalWritable := 'False'} : Bool;   //     Overflow mode error
         OverflowModeWarning { ExternalAccessible := 'False'; ExternalVisible := 'False'; ExternalWritable := 'False'} : Bool;   //     Overflow mode error
         SetDateTimeError { ExternalAccessible := 'False'; ExternalVisible := 'False'; ExternalWritable := 'False'} : Bool;   //     Set date time error
         SetDateTimeWarning { ExternalAccessible := 'False'; ExternalVisible := 'False'; ExternalWritable := 'False'} : Bool;   //     Set date time warning
         InvalidTimeout { ExternalAccessible := 'False'; ExternalVisible := 'False'; ExternalWritable := 'False'} : Bool;   //     Invalid Heartbeat timeout
      END_STRUCT;
      ss_MFCCommand { ExternalAccessible := 'False'; ExternalVisible := 'False'; ExternalWritable := 'False'} : Struct   // MFC command message body for  MessageID = 30020
         Groups { ExternalAccessible := 'False'; ExternalVisible := 'False'; ExternalWritable := 'False'} : Int;
         Nodes { ExternalAccessible := 'False'; ExternalVisible := 'False'; ExternalWritable := 'False'} : Int;
      END_STRUCT;
      st_TimeConverted {InstructionName := 'DTL'; LibVersion := '1.0'; ExternalAccessible := 'False'; ExternalVisible := 'False'; ExternalWritable := 'False'} : DTL;   //   Message date and time converted into DTL data type
      st_PLCTime {InstructionName := 'DTL'; LibVersion := '1.0'; ExternalAccessible := 'False'; ExternalVisible := 'False'; ExternalWritable := 'False'} : DTL;   //   Date and type of the PLC
      sdi_DeserializePosition { ExternalAccessible := 'False'; ExternalVisible := 'False'; ExternalWritable := 'False'} : DInt;   //   Deserialize position
      si_DeserializeHeaderStatus { ExternalAccessible := 'False'; ExternalVisible := 'False'; ExternalWritable := 'False'} : Int;   //   Header deserialize status
      si_DeserializeBodyStatus { ExternalAccessible := 'False'; ExternalVisible := 'False'; ExternalWritable := 'False'} : Int;   //   Body deserialize status
      si_ReadStatus { ExternalAccessible := 'False'; ExternalVisible := 'False'; ExternalWritable := 'False'} : Int;   //   Status of the PLC date and time read operation
      si_WriteStatus { ExternalAccessible := 'False'; ExternalVisible := 'False'; ExternalWritable := 'False'} : Int;   //   Status of the PLC date and time write operation
      si_RingBufferNumber { ExternalAccessible := 'False'; ExternalVisible := 'False'; ExternalWritable := 'False'} : Int := 1;   //   Bad messages ringbuffer counter
      sb_CalculatedChecksum { ExternalAccessible := 'False'; ExternalVisible := 'False'; ExternalWritable := 'False'} : Byte;   //   Calculated checksum
      sx_Heartbeat { ExternalAccessible := 'False'; ExternalVisible := 'False'; ExternalWritable := 'False'} : Bool;   //   Heartbeat message detected
      sx_HeartbeatOK { ExternalAccessible := 'False'; ExternalVisible := 'False'; ExternalWritable := 'False'} : Bool;   //   Heartbeat ok
      sx_SendAllErrorsState { ExternalAccessible := 'False'; ExternalVisible := 'False'; ExternalWritable := 'False'} : Bool;
   END_VAR

   VAR_TEMP
      tx_MessageRead : Bool;   //   Message read from FIFO
      tx_InvalidHeader : Bool;   //   Invalid header
      tx_InvalidMessageID : Bool;   //   Invalid message ID
      tx_BadMessage : Bool;   //   Message with prohibited data
      ti_BadMessageSize : Int;   //   Bad message buffer size
      ti_NumberOfMessageBytes : Int;   //   Length of FIFO message
   END_VAR


BEGIN
	(*
	----------------------------------------------------------------------------------------
	|                                                                                      |
	|  Copyright  2023             FORTNA Europe BV                                        |
	|  All Rights Reserved         Netherlands                                             |
	|                                                                                      |
	----------------------------------------------------------------------------------------
	Version history:
	Date        | Version   | Author       | Remark
	----------------------------------------------------------------------------------------
	03/01/2023  | 1.0       | S. Nikodem   | Release TIA 17 | DHL Munich 2023
	10/08/2023  | 2.0       | M. Diebel    | Send all messages in first connected | DHL Munich 2023
	13/03/2023  | 2.1       | S. Nieswiec  | Updated for new Baseline
	*)


	REGION 1 - Initialize value

	    #sx_SendAllErrorsState := FALSE;

	END_REGION


	REGION 2 – FIFO header status update

	    // Mode 'S' - FIFO register status update.
	    "FC_Fifo"(ic_Mode := 'S',
	              qUDT_Status => #ss_Status.FIFOReceiveStatus,
	              qx_Error => #ss_Status.FIFOReceiveError,
	              qx_Warning => #ss_Status.FIFOReceiveWarning,
	              iqv_Data := #s_UDT_FifoMessage,
	              iqUDT_FifoHeader := #iq_UDT_FifoReceiveHeader,
	              iqv_DataBuffer := #iqs_FifoReceiveData);

	    // FIFO isn't empty and doesn't have error.
	    IF NOT #iq_UDT_FifoReceiveHeader.Status.Empty
	        AND NOT #ss_Status.FIFOReceiveError
	    THEN
	        // Mode 'R' - Read FIFO record.
	        "FC_Fifo"(ic_Mode := 'R',
	                  qUDT_Status => #ss_Status.FIFOReceiveStatus,
	                  qx_Error => #ss_Status.FIFOReceiveError,
	                  qx_Warning => #ss_Status.FIFOReceiveWarning,
	                  iqv_Data := #s_UDT_FifoMessage,
	                  iqUDT_FifoHeader := #iq_UDT_FifoReceiveHeader,
	                  iqv_DataBuffer := #iqs_FifoReceiveData);

	        // Message read bit set.
	        #tx_MessageRead := TRUE;

	        // FIFO empty or FIFO error occured.
	    ELSE
	        #tx_MessageRead := FALSE;
	    END_IF;

	END_REGION

	REGION 3 – Decoding header

	    IF #tx_MessageRead
	    THEN
	        // Converting message header from array of bytes to UDT.
	        #sdi_DeserializePosition := 0;
	        #si_DeserializeHeaderStatus := Deserialize(SRC_ARRAY := #s_UDT_FifoMessage.Bytes,
	                                                   DEST_VARIABLE => #s_UDT_MessageHeader,
	                                                   POS := #sdi_DeserializePosition);
	        REGION 3.1 – Checking checksum

	            "FC_Checksum"(i_UDT_MessageHeader := #s_UDT_MessageHeader,
	                          qb_Checksum => #sb_CalculatedChecksum);

	            // Checking if calculated checksum is valid with checksum in header.
	            IF #sb_CalculatedChecksum <> #s_UDT_MessageHeader.Checksum
	            THEN
	                #tx_InvalidHeader := TRUE;
	            ELSE
	                #tx_InvalidHeader := FALSE;
	            END_IF;

	        END_REGION

	    END_IF;

	END_REGION

	REGION 4 – Message type recognition

	    IF #tx_MessageRead
	        AND NOT #tx_InvalidHeader
	        AND #si_DeserializeHeaderStatus = 0
	    THEN
	        // Invalid message ID initialize.
	        #tx_InvalidMessageID := FALSE;
	        #tx_BadMessage := FALSE;

	        // Heartbeat message.
	        IF #s_UDT_MessageHeader.MessageID = 20
	        THEN
	            #s_UDT_Heartbeat := #s_UDT_MessageHeader;
	            #sx_Heartbeat := TRUE;

	            // Set date time message.
	        ELSIF #s_UDT_MessageHeader.MessageID = 30
	        THEN
	            // Convert array of bytes into body structure
	            #si_DeserializeBodyStatus := Deserialize(SRC_ARRAY := #s_UDT_FifoMessage.Bytes,
	                                                     DEST_VARIABLE => #s_UDT_SetDateTime,
	                                                     POS := #sdi_DeserializePosition);

	            // Date and time validation.
	            IF #s_UDT_SetDateTime.Month >= 1
	                AND #s_UDT_SetDateTime.Month <= 12
	                AND #s_UDT_SetDateTime.Day >= 1
	                AND #s_UDT_SetDateTime.Day <= 31
	                AND #s_UDT_SetDateTime.Hour >= 0
	                AND #s_UDT_SetDateTime.Hour <= 23
	                AND #s_UDT_SetDateTime.Minute >= 0
	                AND #s_UDT_SetDateTime.Minute <= 59
	                AND #s_UDT_SetDateTime.Second >= 0
	                AND #s_UDT_SetDateTime.Second <= 59
	            THEN
	                // Write all others converted components of date and time into the DTL data type variable.
	                #st_TimeConverted.YEAR := INT_TO_UINT(#s_UDT_SetDateTime.Year) + 2000;
	                #st_TimeConverted.MONTH := INT_TO_USINT(#s_UDT_SetDateTime.Month);
	                #st_TimeConverted.DAY := INT_TO_USINT(#s_UDT_SetDateTime.Day);
	                #st_TimeConverted.HOUR := INT_TO_USINT(#s_UDT_SetDateTime.Hour);
	                #st_TimeConverted.MINUTE := INT_TO_USINT(#s_UDT_SetDateTime.Minute);
	                #st_TimeConverted.SECOND := INT_TO_USINT(#s_UDT_SetDateTime.Second);

	                // Read value of the date and time of the PLC and clear the nanoseconds.
	                //#si_ReadStatus := RD_SYS_T(#st_PLCTime);
	                #si_ReadStatus := RD_LOC_T(#st_PLCTime);
	                #st_PLCTime.NANOSECOND := 0;

	                // If the date and time from the message is different then the PLC one change it to the one from message.
	                IF #st_TimeConverted <> #st_PLCTime
	                THEN
	                    //#si_WriteStatus := WR_SYS_T(#st_TimeConverted);
	                    #si_WriteStatus := WR_LOC_T(LOCTIME := #st_TimeConverted, DST := FALSE);

	                END_IF;

	                // Invalid set time message.
	            ELSE
	                #tx_BadMessage := TRUE;
	            END_IF;

	        ELSIF #s_UDT_MessageHeader.MessageID = 30900
	        THEN

	            // Convert array of bytes into structure.
	            #si_DeserializeBodyStatus := Deserialize(SRC_ARRAY := #s_UDT_FifoMessage.Bytes,
	                                                     DEST_VARIABLE => #s_UDT_MFCCommand,
	                                                     POS := #sdi_DeserializePosition);

	            IF #s_UDT_MFCCommand.ClusterID = 2
	                AND #s_UDT_MFCCommand.CommandID = 10
	            THEN
	                #sx_SendAllErrorsState := TRUE;
	            END_IF;

	            // IF #s_UDT_MFCCommand.ClusterID = 1
	            // THEN

	            // IF  #s_UDT_MFCCommand.CommandID = 1
	            // THEN
	            //     "DB_HMICommands".MFCSystemControl.Start := TRUE;

	            // ELSIF #s_UDT_MFCCommand.CommandID = 2
	            // THEN
	            //     "DB_HMICommands".MFCSystemControl.Stop := TRUE;

	            // ELSIF #s_UDT_MFCCommand.CommandID = 3
	            // THEN
	            //     "DB_HMICommands".MFCSystemControl.Reset := TRUE;
	            // END_IF;

	            // END_IF;

	        ELSIF #s_UDT_MessageHeader.MessageID = 30020
	        THEN

	            // Convert array of bytes into structure.
	            #si_DeserializeBodyStatus := Deserialize(SRC_ARRAY := #s_UDT_FifoMessage.Bytes,
	                                                     DEST_VARIABLE => #ss_MFCCommand,
	                                                     POS := #sdi_DeserializePosition);



	            IF #ss_MFCCommand.Groups = 0 AND #ss_MFCCommand.Nodes = 0
	            THEN
	                #sx_SendAllErrorsState := TRUE;
	            END_IF;

	        ELSE
	            // Invalid messsage ID.
	            #tx_InvalidMessageID := TRUE;
	        END_IF;
	    END_IF;

	END_REGION

	REGION 5 - First connection

	    #s_R_TRIG_FirstConnection(CLK := #ix_Connected);


	    IF #s_R_TRIG_FirstConnection.Q AND "DB_MFC_Visu".Configuration.SendAllErrors_FirstConnected
	    THEN

	        #sx_SendAllErrorsState := TRUE;

	    END_IF;

	END_REGION

	REGION 6 – Heartbeat monitoring

	    //HB timeout validation.
	    #ss_Status.InvalidTimeout := #iudi_HeartbeatTimeout <= 0;

	    //HB monitoring if timeout correct.
	    IF NOT #ss_Status.InvalidTimeout
	    THEN
	        #s_R_TRIG_Connected(CLK := #ix_Connected);

	        // Heartbeat timeout monitoring.
	        #s_FB_TimerHeartbeatCheck(iudi_OnDelayTime := 0,
	                                  iudi_OffDelayTime := #iudi_HeartbeatTimeout,
	                                  ix_SignalToDelay := #sx_Heartbeat OR #s_R_TRIG_Connected.Q,
	                                  qx_DelayedSignal => #sx_HeartbeatOK);

	        #sx_Heartbeat := FALSE;
	        #s_F_TRIG_HeartbeatNotOk(CLK := #sx_HeartbeatOK);

	        IF #s_F_TRIG_HeartbeatNotOk.Q
	            AND "DB_Memory".AlwaysFalse
	        THEN
	            // Re-establish conncect with partner and increment the number of communication lost.
	            #iqx_Reconnect := TRUE;
	            #iq_UDT_Statistics.HeartbeatNotObserved += 1;
	        END_IF;
	    END_IF;

	END_REGION

	REGION 7 – Statistics update

	    // Error statistics update required.
	    IF #tx_InvalidHeader
	        OR #tx_InvalidMessageID
	        OR #tx_BadMessage
	    THEN
	        // Invalid message received counter incrementation.
	        #iq_UDT_Statistics.InvalidMessage += 1;

	        // Maximum number of bad messages array.
	        #ti_BadMessageSize := "FC_GetNrOfArrayEl"(#ss_Status.BadMessage);

	        // Writing invalid message in a bad message array.
	        IF #si_RingBufferNumber >= #ti_BadMessageSize
	        THEN
	            #si_RingBufferNumber := 1;
	        END_IF;

	        #ti_NumberOfMessageBytes := "FC_GetNrOfArrayEl"(iv_Array := #s_UDT_FifoMessage.Bytes);

	        MOVE_BLK(IN := #s_UDT_FifoMessage.Bytes[0],
	                 COUNT := INT_TO_UINT(#ti_NumberOfMessageBytes) - 1,
	                 OUT => #ss_Status.BadMessage[#si_RingBufferNumber].Bytes[0]);

	        #si_RingBufferNumber += 1;
	    END_IF;

	    //Resetting statistics.
	    IF #ix_ResetData
	    THEN
	        #iq_UDT_Statistics.InvalidMessage := 0;
	        #iq_UDT_Statistics.HeartbeatNotObserved := 0;
	    END_IF;

	END_REGION

	REGION 9 – Status

	    // Collective error output.
	    #qx_Error :=
	    #ss_Status.FIFOReceiveError
	    OR #ss_Status.InvalidTimeout
	    OR #ss_Status.SetDateTimeError
	    OR #ss_Status.OverflowModeError
	    OR #ss_Status.OperationModeError;

	    // Collective warning output.
	    #qx_Warning :=
	    #ss_Status.FIFOReceiveWarning
	    OR #ss_Status.OperationModeWarning
	    OR #ss_Status.OverflowModeWarning
	    OR #ss_Status.SetDateTimeWarning;

	END_REGION

	REGION Write Output

	    #qx_SendAllErrorsState := #sx_SendAllErrorsState;

	END_REGION
END_FUNCTION_BLOCK

FUNCTION_BLOCK "FB_MFC_Visu_Rapiscan_Status"
{ S7_Optimized_Access := 'TRUE' }
VERSION : 0.1
// ATTRIBUTES
// AUTO_NUMBER = True
// BLOCK_NUMBER = 156
// END_ATTRIBUTES
   VAR_INPUT
      i_UDT_RapiscanStatus { ExternalAccessible := 'False'; ExternalVisible := 'False'; ExternalWritable := 'False'} : "UDT_RapiscanStatus";   // Rapiscan status structure
      i_UDT_EquipmentNumber { ExternalAccessible := 'False'; ExternalVisible := 'False'; ExternalWritable := 'False'} : "UDT_EquipmentNumber";   // Item number
      ix_SendAllErrorsState { ExternalAccessible := 'False'; ExternalVisible := 'False'; ExternalWritable := 'False'} : Bool;   // True - update all the messages
      ix_MFCConnected { ExternalAccessible := 'False'; ExternalVisible := 'False'; ExternalWritable := 'False'} : Bool;   // True - A connection to the MFC has been established
      ix_CollectiveReset { ExternalAccessible := 'False'; ExternalVisible := 'False'; ExternalWritable := 'False'} : Bool;   // True - Collective reset command of all system controls
   END_VAR

   VAR_OUTPUT
      qx_Error { ExternalAccessible := 'False'; ExternalVisible := 'False'; ExternalWritable := 'False'} : Bool;   // Block error
      qx_Warning { ExternalAccessible := 'False'; ExternalVisible := 'False'; ExternalWritable := 'False'} : Bool;   // Block warning
   END_VAR

   VAR_IN_OUT
      iq_UDT_FifoHeader : "UDT_FifoHeader";   // FIFO header
      iqs_FifoData : Array[*] of "UDT_MessageV2";   // FIFO data buffer
      iqdi_MessageSequenceNumber { ExternalAccessible := 'False'; ExternalVisible := 'False'; ExternalWritable := 'False'} : DInt;   // Message number
   END_VAR

   VAR
      s_FB_ItemError { ExternalAccessible := 'False'; ExternalVisible := 'False'; ExternalWritable := 'False'; S7_SetPoint := 'False'} : "FB_ItemError";   // Item error block's instance
      s_FB_ItemStatus { ExternalAccessible := 'False'; ExternalVisible := 'False'; ExternalWritable := 'False'; S7_SetPoint := 'False'} : "FB_ItemStatus";   // Item status block's instance
      ss_FIFOStatus { ExternalAccessible := 'False'; ExternalVisible := 'False'; ExternalWritable := 'False'; S7_SetPoint := 'False'} : "UDT_FifoStatus";   // Status structure
      s_UDT_Message { ExternalAccessible := 'False'; ExternalVisible := 'False'; ExternalWritable := 'False'; S7_SetPoint := 'False'} : "UDT_MessageV2";   // Message
      s_UDT_RapiscanOld { ExternalAccessible := 'False'; ExternalVisible := 'False'; ExternalWritable := 'False'; S7_SetPoint := 'False'} : "UDT_RapiscanStatus";   // Rapiscan status structure
      s_UDT_ItemError { ExternalAccessible := 'False'; ExternalVisible := 'False'; ExternalWritable := 'False'; S7_SetPoint := 'False'} : "UDT_ItemError";   // Item error message body structure
      s_UDT_ItemStatus { ExternalAccessible := 'False'; ExternalVisible := 'False'; ExternalWritable := 'False'; S7_SetPoint := 'False'} : "UDT_ItemStatus";   // Item status message body structure
      s_R_TRIG_Connection {InstructionName := 'R_TRIG'; LibVersion := '1.0'; ExternalAccessible := 'False'; ExternalVisible := 'False'; ExternalWritable := 'False'; S7_SetPoint := 'False'} : R_TRIG;   // Rising edge trigger connection reastablished
      s_F_TRIG_SendAllErrors {InstructionName := 'F_TRIG'; LibVersion := '1.0'; ExternalAccessible := 'False'; ExternalVisible := 'False'; ExternalWritable := 'False'; S7_SetPoint := 'False'} : F_TRIG;   // Falling edge trigger from signal send all errors
      sdi_Code { ExternalAccessible := 'False'; ExternalVisible := 'False'; ExternalWritable := 'False'} : DInt;   // Error code
      si_ItemStatus { ExternalAccessible := 'False'; ExternalVisible := 'False'; ExternalWritable := 'False'} : Int;   // Item status
      ii_ErrorNumber { ExternalAccessible := 'False'; ExternalVisible := 'False'; ExternalWritable := 'False'} : Int;   // Counter Error Number
      si_State { ExternalAccessible := 'False'; ExternalVisible := 'False'; ExternalWritable := 'False'} : Int;   // Error state
      sx_ItemErrorMessageReq { ExternalAccessible := 'False'; ExternalVisible := 'False'; ExternalWritable := 'False'} : Bool;   // Item error message required
      sx_ItemStatusMessageReq { ExternalAccessible := 'False'; ExternalVisible := 'False'; ExternalWritable := 'False'} : Bool;   // Item status message required
      sx_SendAllProcedure { ExternalAccessible := 'False'; ExternalVisible := 'False'; ExternalWritable := 'False'} : Bool;   // Send all procedure
      sx_FIFOError { ExternalAccessible := 'False'; ExternalVisible := 'False'; ExternalWritable := 'False'} : Bool;   // FIFO error
      sx_FIFOWarning { ExternalAccessible := 'False'; ExternalVisible := 'False'; ExternalWritable := 'False'} : Bool;   // FIFO warning
      sx_ItemErrorBlockError { ExternalAccessible := 'False'; ExternalVisible := 'False'; ExternalWritable := 'False'} : Bool;   // Item error block error
      sx_ItemErrorBlockWarning { ExternalAccessible := 'False'; ExternalVisible := 'False'; ExternalWritable := 'False'} : Bool;   // Item error block warning
      sx_ItemStatusBlockError { ExternalAccessible := 'False'; ExternalVisible := 'False'; ExternalWritable := 'False'} : Bool;   // Item status block error
      sx_ItemStatusBlockWarning { ExternalAccessible := 'False'; ExternalVisible := 'False'; ExternalWritable := 'False'} : Bool;   // Item status block warning
   END_VAR


BEGIN
	(*
	----------------------------------------------------------------------------------------
	|                                                                                      |
	|  Copyright  2023             FORTNA Europe BV                                        |
	|  All Rights Reserved         Netherlands                                             |
	|                                                                                      |
	----------------------------------------------------------------------------------------
	Version history:
	Date        | Version   | Author       | Remark
	----------------------------------------------------------------------------------------
	27/03/2023  | 1.0       | M. Diebel   | Release TIA 17 | DHL Munich 2023
	13/03/2023  | 1.1       | S. Nieswiec | Updated for new Baseline
	*)


	REGION 1 - Initialize message required signals

	    #sx_ItemErrorMessageReq := FALSE;
	    #sx_ItemStatusMessageReq := FALSE;

	    // On connection reestablish send last remembered status and error state ( status only when it's diffrent then 0 )
	    #s_R_TRIG_Connection(CLK := #ix_MFCConnected);

	    IF #s_R_TRIG_Connection.Q AND #si_ItemStatus <> 0
	    THEN
	        #sx_ItemStatusMessageReq := TRUE;
	    END_IF;

	    IF #s_R_TRIG_Connection.Q
	    THEN
	        #sx_ItemErrorMessageReq := TRUE;
	    END_IF;

	    // Prepare trigger on the collective reset signal.
	    #s_F_TRIG_SendAllErrors(CLK := #ix_SendAllErrorsState);

	    // When collective reset will go down, start send every equipment errors.
	    IF #s_F_TRIG_SendAllErrors.Q AND NOT #sx_SendAllProcedure
	    THEN
	        #ii_ErrorNumber := 0;
	        #sx_SendAllProcedure := TRUE;
	    END_IF;

	END_REGION

	REGION 2 - FIFO header status update

	    // Mode 'S' - FIFO register status update.
	    "FC_Fifo"(ic_Mode := 'S',
	              qUDT_Status => #ss_FIFOStatus,
	              qx_Error => #sx_FIFOError,
	              qx_Warning => #sx_FIFOWarning,
	              iqv_Data := #s_UDT_Message,
	              iqUDT_FifoHeader := #iq_UDT_FifoHeader,
	              iqv_DataBuffer := #iqs_FifoData);

	END_REGION

	REGION 3 - Prepare message data

	    // When there is no reset errors command, update status and errors.
	    IF NOT #ix_CollectiveReset
	        AND NOT #ss_FIFOStatus.FifoPreFull
	    THEN
	        // Status
	        IF (#i_UDT_RapiscanStatus.Status <> #s_UDT_RapiscanOld.Status OR (#sx_SendAllProcedure AND #ii_ErrorNumber = 0))
	        THEN
	            #sx_ItemStatusMessageReq := TRUE;
	            #si_ItemStatus := #i_UDT_RapiscanStatus.Status;
	            #s_UDT_RapiscanOld.Status := #i_UDT_RapiscanStatus.Status;
	        END_IF;


	        // Check which specific status changed, prepare code, change state and write new status into the old one.
	        IF (#i_UDT_RapiscanStatus.XraySpecific.XrayEnergised <> #s_UDT_RapiscanOld.XraySpecific.XrayEnergised AND NOT #sx_SendAllProcedure)
	            OR (#sx_SendAllProcedure AND #ii_ErrorNumber = 0)
	        THEN
	            #sdi_Code := "DB_MFC_ErrorCode".Rapiscan.XrayEnergised;
	            #si_State := BOOL_TO_INT(#i_UDT_RapiscanStatus.XraySpecific.XrayEnergised);
	            #s_UDT_RapiscanOld.XraySpecific.XrayEnergised := #i_UDT_RapiscanStatus.XraySpecific.XrayEnergised;
	            #sx_ItemErrorMessageReq := TRUE;
	            #ii_ErrorNumber += 1;
	        ELSIF (#i_UDT_RapiscanStatus.XraySpecific.XrayFault <> #s_UDT_RapiscanOld.XraySpecific.XrayFault AND NOT #sx_SendAllProcedure)
	            OR (#sx_SendAllProcedure AND #ii_ErrorNumber = 1)
	        THEN
	            #sdi_Code := "DB_MFC_ErrorCode".Rapiscan.XrayFault;
	            #si_State := BOOL_TO_INT(#i_UDT_RapiscanStatus.XraySpecific.XrayFault);
	            #s_UDT_RapiscanOld.XraySpecific.XrayFault := #i_UDT_RapiscanStatus.XraySpecific.XrayFault;
	            #sx_ItemErrorMessageReq := TRUE;
	            #ii_ErrorNumber += 1;
	        ELSIF (#i_UDT_RapiscanStatus.XraySpecific.XrayRdyRCV <> #s_UDT_RapiscanOld.XraySpecific.XrayRdyRCV AND NOT #sx_SendAllProcedure)
	            OR (#sx_SendAllProcedure AND #ii_ErrorNumber = 2)
	        THEN
	            #sdi_Code := "DB_MFC_ErrorCode".Rapiscan.XrayRdyRCV;
	            #si_State := BOOL_TO_INT(#i_UDT_RapiscanStatus.XraySpecific.XrayRdyRCV);
	            #s_UDT_RapiscanOld.XraySpecific.XrayRdyRCV := #i_UDT_RapiscanStatus.XraySpecific.XrayRdyRCV;
	            #sx_ItemErrorMessageReq := TRUE;
	            #ii_ErrorNumber += 1;
	        ELSIF (#i_UDT_RapiscanStatus.XraySpecific.XrayRdySend <> #s_UDT_RapiscanOld.XraySpecific.XrayRdySend AND NOT #sx_SendAllProcedure)
	            OR (#sx_SendAllProcedure AND #ii_ErrorNumber = 3)
	        THEN
	            #sdi_Code := "DB_MFC_ErrorCode".Rapiscan.XrayRdySend;
	            #si_State := BOOL_TO_INT(#i_UDT_RapiscanStatus.XraySpecific.XrayRdySend);
	            #s_UDT_RapiscanOld.XraySpecific.XrayRdySend := #i_UDT_RapiscanStatus.XraySpecific.XrayRdySend;
	            #sx_ItemErrorMessageReq := TRUE;
	            #ii_ErrorNumber += 1;
	        ELSIF (#i_UDT_RapiscanStatus.XraySpecific.BagScanning <> #s_UDT_RapiscanOld.XraySpecific.BagScanning AND NOT #sx_SendAllProcedure)
	            OR (#sx_SendAllProcedure AND #ii_ErrorNumber = 4)
	        THEN
	            #sdi_Code := "DB_MFC_ErrorCode".Rapiscan.BagScanning;
	            #si_State := BOOL_TO_INT(#i_UDT_RapiscanStatus.XraySpecific.BagScanning);
	            #s_UDT_RapiscanOld.XraySpecific.BagScanning := #i_UDT_RapiscanStatus.XraySpecific.BagScanning;
	            #sx_ItemErrorMessageReq := TRUE;
	            #ii_ErrorNumber += 1;
	        ELSIF (#i_UDT_RapiscanStatus.XraySpecific.TransportMode <> #s_UDT_RapiscanOld.XraySpecific.TransportMode AND NOT #sx_SendAllProcedure)
	            OR (#sx_SendAllProcedure AND #ii_ErrorNumber = 5)
	        THEN
	            #sdi_Code := "DB_MFC_ErrorCode".Rapiscan.TransportMode;
	            #si_State := BOOL_TO_INT(#i_UDT_RapiscanStatus.XraySpecific.TransportMode);
	            #s_UDT_RapiscanOld.XraySpecific.TransportMode := #i_UDT_RapiscanStatus.XraySpecific.TransportMode;
	            #sx_ItemErrorMessageReq := TRUE;
	            #ii_ErrorNumber += 1;
	        ELSIF (#i_UDT_RapiscanStatus.XraySpecific.BackBelt <> #s_UDT_RapiscanOld.XraySpecific.BackBelt AND NOT #sx_SendAllProcedure)
	            OR (#sx_SendAllProcedure AND #ii_ErrorNumber = 6)
	        THEN
	            #sdi_Code := "DB_MFC_ErrorCode".Rapiscan.BackBelt;
	            #si_State := BOOL_TO_INT(#i_UDT_RapiscanStatus.XraySpecific.BackBelt);
	            #s_UDT_RapiscanOld.XraySpecific.BackBelt := #i_UDT_RapiscanStatus.XraySpecific.BackBelt;
	            #sx_ItemErrorMessageReq := TRUE;
	            #sx_SendAllProcedure := FALSE;
	            #ii_ErrorNumber += 1;
	        END_IF;
	    END_IF;
	END_REGION

	REGION 4 - Write message components to the item error structure

	    #s_UDT_ItemError.ItemNumber := #i_UDT_EquipmentNumber;
	    #s_UDT_ItemError.Error := #sdi_Code;
	    #s_UDT_ItemError.State := #si_State;
	    #s_UDT_ItemError.Masked := 1;

	END_REGION

	REGION 5 - Write message components to the item status structure

	    #s_UDT_ItemStatus.Group := #i_UDT_EquipmentNumber.Group;
	    #s_UDT_ItemStatus.Node := #i_UDT_EquipmentNumber.Node;
	    #s_UDT_ItemStatus.Status := #si_ItemStatus;

	END_REGION

	REGION 6 - Prepare messages to the MFC

	    // If item error message required signal is set, prepare the item error message.
	    IF (#sx_ItemErrorMessageReq)
	    THEN
	        #s_FB_ItemError(i_UDT_ItemErrorBody := #s_UDT_ItemError,
	                        ii_MessageGroup := 1,
	                        ix_FlagRetry := FALSE,
	                        idi_TimeSpan := 0,
	                        qx_Error => #sx_ItemErrorBlockError,
	                        qx_Warning => #sx_ItemErrorBlockWarning,
	                        iq_UDT_FifoHeader := #iq_UDT_FifoHeader,
	                        iqs_FifoData := #iqs_FifoData,
	                        iqdi_MessageSequenceNumber := #iqdi_MessageSequenceNumber);
	    END_IF;

	    // If item status message required signal is set, prepare the item error message.
	    IF (#sx_ItemStatusMessageReq)
	    THEN
	        #s_FB_ItemStatus(i_UDT_ItemStatusBody := #s_UDT_ItemStatus,
	                         ii_MessageGroup := 1,
	                         ix_FlagRetry := FALSE,
	                         idi_TimeSpan := 0,
	                         qx_Error => #sx_ItemStatusBlockError,
	                         qx_Warning => #sx_ItemStatusBlockWarning,
	                         iq_UDT_FifoHeader := #iq_UDT_FifoHeader,
	                         iqs_FifoData := #iqs_FifoData,
	                         iqdi_MessageSequenceNumber := #iqdi_MessageSequenceNumber);
	    END_IF;

	END_REGION

	REGION 7 - Write outputs

	    // Prepare collective output error.
	    #qx_Error :=
	    #sx_ItemErrorBlockError
	    OR #sx_ItemStatusBlockError
	    OR #sx_FIFOError;

	    // Prepare collective output warning.
	    #qx_Warning :=
	    #sx_ItemErrorBlockWarning
	    OR #sx_ItemStatusBlockWarning
	    OR #sx_FIFOWarning;

	END_REGION

END_FUNCTION_BLOCK

FUNCTION_BLOCK "FB_MessageCompresion"
{ S7_Optimized_Access := 'TRUE' }
VERSION : 2.0
// ATTRIBUTES
// AUTO_NUMBER = True
// BLOCK_NUMBER = 133
// END_ATTRIBUTES
   VAR_IN_OUT
      iq_UDT_FifoReceiveHeader_In : "UDT_FifoHeader";   // Data to be compressed - Fifo Header
      iqs_FifoReceiveData_In : Array[*] of "UDT_MessageV2";   // Data to be compressed - Fiffo Data
      iqdi_MessageSequenceNumber { ExternalAccessible := 'False'; ExternalVisible := 'False'; ExternalWritable := 'False'} : DInt;   // Message number
      iq_UDT_FifoReceiveHeader_Out : "UDT_FifoHeader";   // Data compressed - Fifo Header
      iqs_FifoReceiveData_Out : Array[*] of "UDT_MessageV2";   // Data compressed - Fiffo Data
   END_VAR

   VAR
      s_UDT_MessageHeader { ExternalAccessible := 'False'; ExternalVisible := 'False'; ExternalWritable := 'False'; S7_SetPoint := 'False'} : "UDT_MessageHeaderV2";   // Message header
      s_UDT_FifoMessage { ExternalAccessible := 'False'; ExternalVisible := 'False'; ExternalWritable := 'False'; S7_SetPoint := 'False'} : "UDT_MessageV2";
      s_UDT_MessageArray { ExternalAccessible := 'False'; ExternalVisible := 'False'; ExternalWritable := 'False'; S7_SetPoint := 'False'} : "UDT_MessageV2";
      s_UDT_MessageArray_Empty { ExternalAccessible := 'False'; ExternalVisible := 'False'; ExternalWritable := 'False'; S7_SetPoint := 'False'} : "UDT_MessageV2";
      s_UDT_ItemErrorBody { ExternalAccessible := 'False'; ExternalVisible := 'False'; ExternalWritable := 'False'; S7_SetPoint := 'False'} : "UDT_ItemError";   // Item error message body structure
      s_UDT_ItemStatusBody { ExternalAccessible := 'False'; ExternalVisible := 'False'; ExternalWritable := 'False'; S7_SetPoint := 'False'} : "UDT_ItemStatus";   // Item status message body structure
      sa_Data_ItemError { ExternalAccessible := 'False'; ExternalVisible := 'False'; ExternalWritable := 'False'; S7_SetPoint := 'False'} : Array[0..1001] of "UDT_ItemError";
      sa_Data_ItemStatus { ExternalAccessible := 'False'; ExternalVisible := 'False'; ExternalWritable := 'False'; S7_SetPoint := 'False'} : Array[0..1001] of "UDT_ItemStatus";
      sa_Data_InvalidMessageID { ExternalAccessible := 'False'; ExternalVisible := 'False'; ExternalWritable := 'False'; S7_SetPoint := 'False'} : Array[0..1001] of "UDT_MessageV2";
      ss_NewErrorMessage { ExternalAccessible := 'False'; ExternalVisible := 'False'; ExternalWritable := 'False'} : Array[0..101] of Struct
         Size { ExternalAccessible := 'False'; ExternalVisible := 'False'; ExternalWritable := 'False'} : Int;
         Body { ExternalAccessible := 'False'; ExternalVisible := 'False'; ExternalWritable := 'False'; S7_SetPoint := 'False'} : Array[1..100] of "UDT_ItemError";
      END_STRUCT;
      ss_NewStatusMessage { ExternalAccessible := 'False'; ExternalVisible := 'False'; ExternalWritable := 'False'} : Array[0..101] of Struct
         Size { ExternalAccessible := 'False'; ExternalVisible := 'False'; ExternalWritable := 'False'} : Int;
         Body { ExternalAccessible := 'False'; ExternalVisible := 'False'; ExternalWritable := 'False'; S7_SetPoint := 'False'} : Array[1..1000] of "UDT_ItemStatus";
      END_STRUCT;
      ss_NewErrorMessage_Empty { ExternalAccessible := 'False'; ExternalVisible := 'False'; ExternalWritable := 'False'} : Array[0..101] of Struct
         Size { ExternalAccessible := 'False'; ExternalVisible := 'False'; ExternalWritable := 'False'} : Int;
         Body { ExternalAccessible := 'False'; ExternalVisible := 'False'; ExternalWritable := 'False'; S7_SetPoint := 'False'} : Array[1..100] of "UDT_ItemError";
      END_STRUCT;
      ss_NewStatusMessage_Empty { ExternalAccessible := 'False'; ExternalVisible := 'False'; ExternalWritable := 'False'} : Array[0..101] of Struct
         Size { ExternalAccessible := 'False'; ExternalVisible := 'False'; ExternalWritable := 'False'} : Int;
         Body { ExternalAccessible := 'False'; ExternalVisible := 'False'; ExternalWritable := 'False'; S7_SetPoint := 'False'} : Array[1..1000] of "UDT_ItemStatus";
      END_STRUCT;
      ss_Status { ExternalAccessible := 'False'; ExternalVisible := 'False'; ExternalWritable := 'False'} : Struct   // Status structure - Fifo
         FIFOReceiveStatus { ExternalAccessible := 'False'; ExternalVisible := 'False'; ExternalWritable := 'False'} : "UDT_FifoStatus";
         FIFOInvalidMessageIDStatus { ExternalAccessible := 'False'; ExternalVisible := 'False'; ExternalWritable := 'False'} : "UDT_FifoStatus";
         FIFOItemErrorStatus { ExternalAccessible := 'False'; ExternalVisible := 'False'; ExternalWritable := 'False'} : "UDT_FifoStatus";
         FIFOItemStatusStatus { ExternalAccessible := 'False'; ExternalVisible := 'False'; ExternalWritable := 'False'} : "UDT_FifoStatus";
         FIFOError { ExternalAccessible := 'False'; ExternalVisible := 'False'; ExternalWritable := 'False'; S7_SetPoint := 'True'} : Bool;   //   FIFO error
         FIFOWarning { ExternalAccessible := 'False'; ExternalVisible := 'False'; ExternalWritable := 'False'; S7_SetPoint := 'True'} : Bool;   //   FIFO warning
         InvalidMessageArraySize { ExternalAccessible := 'False'; ExternalVisible := 'False'; ExternalWritable := 'False'} : Bool;   //   Message array is too short for message
      END_STRUCT;
      sdi_DeserializePosition { ExternalAccessible := 'False'; ExternalVisible := 'False'; ExternalWritable := 'False'} : DInt;   // Deserialize position
      si_DeserializeHeaderStatus { ExternalAccessible := 'False'; ExternalVisible := 'False'; ExternalWritable := 'False'} : Int;   // Header deserialize status
      sb_CalculatedChecksum { ExternalAccessible := 'False'; ExternalVisible := 'False'; ExternalWritable := 'False'} : Byte;   // Calculated checksum
      si_DeserializeBodyStatus { ExternalAccessible := 'False'; ExternalVisible := 'False'; ExternalWritable := 'False'} : Int;   // Body deserialize status
      si_Counter_ItemError { ExternalAccessible := 'False'; ExternalVisible := 'False'; ExternalWritable := 'False'} : Int := 0;
      si_Counter_ItemStatus { ExternalAccessible := 'False'; ExternalVisible := 'False'; ExternalWritable := 'False'} : Int := 0;
      si_Counter_InvalidMessageID { ExternalAccessible := 'False'; ExternalVisible := 'False'; ExternalWritable := 'False'} : Int := 0;
      si_ItemError_MessageToCompress { ExternalAccessible := 'False'; ExternalVisible := 'False'; ExternalWritable := 'False'} : Int;
      si_NewMessage_Counter { ExternalAccessible := 'False'; ExternalVisible := 'False'; ExternalWritable := 'False'} : Int;
      si_StoredMessages { ExternalAccessible := 'False'; ExternalVisible := 'False'; ExternalWritable := 'False'} : Int;
      si_HeaderSerializeStatus { ExternalAccessible := 'False'; ExternalVisible := 'False'; ExternalWritable := 'False'} : Int;
      si_BodySerializeStatus { ExternalAccessible := 'False'; ExternalVisible := 'False'; ExternalWritable := 'False'} : Int;
      sdi_SerializePosition { ExternalAccessible := 'False'; ExternalVisible := 'False'; ExternalWritable := 'False'} : DInt;
      si_BodyLenght { ExternalAccessible := 'False'; ExternalVisible := 'False'; ExternalWritable := 'False'} : Int;
      test { ExternalAccessible := 'False'; ExternalVisible := 'False'; ExternalWritable := 'False'} : Array[0..1000] of Int;
   END_VAR

   VAR_TEMP
      tx_MessageRead : Bool;   // Message read correctly
      tx_InvalidHeader : Bool;   // Invalid header
      ti_Loop_CopyData : Int;   // Loop counter - Copy data from Fifo
      ti_Loop_InvalidMessageID : Int;   // Loop counter - Write data to Fifo
      ti_Loop_ItemError : Int;   // Loop counter - Write data to Fifo
      ti_Loop_ItemError_FiFo : Int;
      ti_Loop_ItemError_FiFo_1 : Int;
      ti_Loop_ItemStatus_FiFo : Int;
      ti_Loop_ItemStatus_FiFo_1 : Int;
      ti_Loop_ItemStatus : Int;   // Loop counter - Write data to Fifo
   END_VAR

   VAR CONSTANT
      ci_ItemStatus_MessageLength : Int := 24;   // Message length in bytes
      ci_ItemStatus_BodyLenght : Int := 6;   // Message body length
      ci_ItemError_MessageLenght : Int := 34;   // Message length in bytes
      ci_ItemError_BodyLenght : Int := 16;   // Message body length
      ci_ItemError_BodyMaxSize : Int := 16;
      ci_ItemStatus_BodyMaxSize : Int := 12;
      ci_ItemStatus_MessageID : Int := 21020;   // Message ID number
      ci_ItemError_MessageID : Int := 21010;   // Message ID number
   END_VAR


BEGIN
	(*
	----------------------------------------------------------------------------------------
	|                                                                                      |
	|  Copyright  2023             FORTNA Europe BV                                        |
	|  All Rights Reserved         Netherlands                                             |
	|                                                                                      |
	----------------------------------------------------------------------------------------

	Version history:
	Date        | Version   | Author       | Remark
	----------------------------------------------------------------------------------------
	21/12/2022  | 1.0       | S. Nikodem   | Release TIA 17 | DHL Munich 2023
	11/08/2023  | 2.0       | M. Diebel    | Fixed issues   | DHL Munich 2023
	05/03/2024  | 2.1       | M. Diebel    | Cleas message data   | DHL Munich 2023
	13/03/2023  | 2.2       | S. Nieswiec  | Updated for new Baseline
	*)


	REGION 1 - Deactivate the function

	    //When are less like 2 messages in the array
	    IF #iq_UDT_FifoReceiveHeader_In.TotalEntriesStored < 2 THEN

	        RETURN;
	    END_IF;

	END_REGION

	REGION 2 - Copy data
	    //Copy data from FiFo to static memory

	    //Set how many message take to array from FIFO
	    #si_StoredMessages := "DB_MFC_Visu".Configuration.NumberOfCompressedMessages;

	    //Initial value
	    #si_Counter_ItemError := 0;
	    #si_Counter_ItemStatus := 0;
	    #si_Counter_InvalidMessageID := 0;

	    FOR #ti_Loop_CopyData := 1 TO #si_StoredMessages DO

	        REGION 2.1 – FIFO

	            // Mode 'S' - FIFO register status update.
	            "FC_Fifo"(ic_Mode := 'S',
	                      qUDT_Status => #ss_Status.FIFOReceiveStatus,
	                      qx_Error => #ss_Status.FIFOError,
	                      qx_Warning => #ss_Status.FIFOWarning,
	                      iqv_Data := #s_UDT_FifoMessage,
	                      iqUDT_FifoHeader := #iq_UDT_FifoReceiveHeader_In,
	                      iqv_DataBuffer := #iqs_FifoReceiveData_In);

	            // FIFO isn't empty and doesn't have error.
	            IF NOT #iq_UDT_FifoReceiveHeader_In.Status.Empty
	                AND NOT #ss_Status.FIFOError
	            THEN
	                // Mode 'R' - Read FIFO record.
	                "FC_Fifo"(ic_Mode := 'R',
	                          qUDT_Status => #ss_Status.FIFOReceiveStatus,
	                          qx_Error => #ss_Status.FIFOError,
	                          qx_Warning => #ss_Status.FIFOWarning,
	                          iqv_Data := #s_UDT_FifoMessage,
	                          iqUDT_FifoHeader := #iq_UDT_FifoReceiveHeader_In,
	                          iqv_DataBuffer := #iqs_FifoReceiveData_In);

	                // Message read bit set.
	                #tx_MessageRead := TRUE;
	            ELSE
	                #tx_MessageRead := FALSE;
	            END_IF;

	        END_REGION

	        REGION 2.2 – Decoding header

	            IF #tx_MessageRead
	            THEN
	                // Converting message header from array of bytes to UDT.
	                #sdi_DeserializePosition := 0;
	                #si_DeserializeHeaderStatus := Deserialize(SRC_ARRAY := #s_UDT_FifoMessage.Bytes,
	                                                           DEST_VARIABLE => #s_UDT_MessageHeader,
	                                                           POS := #sdi_DeserializePosition);

	                //Checking checksum
	                "FC_Checksum"(i_UDT_MessageHeader := #s_UDT_MessageHeader,
	                              qb_Checksum => #sb_CalculatedChecksum);

	                // Checking if calculated checksum is valid with checksum in header.
	                IF #sb_CalculatedChecksum <> #s_UDT_MessageHeader.Checksum
	                THEN
	                    #tx_InvalidHeader := TRUE;
	                ELSE
	                    #tx_InvalidHeader := FALSE;
	                END_IF;

	            END_IF;

	        END_REGION

	        REGION 2.3 – Message type recognition

	            IF #tx_MessageRead
	                AND NOT #tx_InvalidHeader
	                AND #si_DeserializeHeaderStatus = 0
	            THEN

	                //Item error message.
	                IF #s_UDT_MessageHeader.MessageID = #ci_ItemError_MessageID AND #s_UDT_MessageHeader.BodyLength = #ci_ItemError_BodyLenght
	                THEN
	                    // Convert array of bytes into body structure.
	                    #si_DeserializeBodyStatus := Deserialize(SRC_ARRAY := #s_UDT_FifoMessage.Bytes,
	                                                             DEST_VARIABLE => #s_UDT_ItemErrorBody,
	                                                             POS := #sdi_DeserializePosition);
	                    //Add up position
	                    #si_Counter_ItemError += 1;
	                    //Copy data to array
	                    #sa_Data_ItemError[#si_Counter_ItemError] := #s_UDT_ItemErrorBody;


	                    // Item status message.
	                ELSIF #s_UDT_MessageHeader.MessageID = #ci_ItemStatus_MessageID AND #s_UDT_MessageHeader.BodyLength = #ci_ItemStatus_BodyLenght
	                THEN
	                    // Convert array of bytes into body structure.
	                    #si_DeserializeBodyStatus := Deserialize(SRC_ARRAY := #s_UDT_FifoMessage.Bytes,
	                                                             DEST_VARIABLE => #s_UDT_ItemStatusBody,
	                                                             POS := #sdi_DeserializePosition);
	                    //Add up position
	                    #si_Counter_ItemStatus += 1;
	                    //Copy data to array
	                    #sa_Data_ItemStatus[#si_Counter_ItemStatus] := #s_UDT_ItemStatusBody;

	                ELSE

	                    //Add up position
	                    #si_Counter_InvalidMessageID += 1;
	                    //Copy data to array
	                    #sa_Data_InvalidMessageID[#si_Counter_InvalidMessageID] := #s_UDT_FifoMessage;

	                END_IF;

	            END_IF;

	        END_REGION

	    END_FOR;

	END_REGION

	REGION 3 - Crate new message

	    REGION 3.1 - Item Error

	        IF #si_Counter_ItemError >= 1 THEN

	            #si_NewMessage_Counter := 1;
	            #ss_NewErrorMessage := #ss_NewErrorMessage_Empty;
	            #s_UDT_MessageArray.Bytes := #s_UDT_MessageArray_Empty.Bytes;

	            // Crate new messages
	            FOR #ti_Loop_ItemError := 1 TO #si_Counter_ItemError DO

	                IF #ss_NewErrorMessage[#si_NewMessage_Counter].Size > #ci_ItemError_BodyMaxSize THEN

	                    #si_NewMessage_Counter += 1;

	                END_IF;

	                #ss_NewErrorMessage[#si_NewMessage_Counter].Body[#ti_Loop_ItemError] := #sa_Data_ItemError[#ti_Loop_ItemError];
	                #ss_NewErrorMessage[#si_NewMessage_Counter].Size += 1;

	            END_FOR;


	            FOR #ti_Loop_ItemError_FiFo := 1 TO #si_NewMessage_Counter DO

	                // Check sequence number. If it is equal or greater than 30000 reset it to 1.
	                IF #iqdi_MessageSequenceNumber < 30000
	                THEN
	                    #iqdi_MessageSequenceNumber += 1;
	                ELSE
	                    #iqdi_MessageSequenceNumber := 1;
	                END_IF;

	                #ss_NewErrorMessage[#ti_Loop_ItemError_FiFo].Size := #ss_NewErrorMessage[#ti_Loop_ItemError_FiFo].Size * #ci_ItemError_BodyLenght;

	                // Write parts of the header into structure.
	                #s_UDT_MessageHeader.BodyLength := #ss_NewErrorMessage[#ti_Loop_ItemError_FiFo].Size;
	                #s_UDT_MessageHeader.FlagRetry.%X0 := FALSE;
	                #s_UDT_MessageHeader.Group := 1;
	                #s_UDT_MessageHeader.MessageID := #ci_ItemError_MessageID;
	                #s_UDT_MessageHeader.SequenceNumber := #iqdi_MessageSequenceNumber;
	                #s_UDT_MessageHeader.TimeSpan := 0;

	                // Calculate the header checksum.
	                "FC_Checksum"(i_UDT_MessageHeader := #s_UDT_MessageHeader,
	                              qb_Checksum => #s_UDT_MessageHeader.Checksum);


	                // Initialize the header serialize position and convert header structure into array of bytes.
	                #sdi_SerializePosition := 0;
	                #si_HeaderSerializeStatus := Serialize(SRC_VARIABLE := #s_UDT_MessageHeader,
	                                                       DEST_ARRAY => #s_UDT_MessageArray.Bytes,
	                                                       POS := #sdi_SerializePosition);

	                FOR #ti_Loop_ItemError_FiFo_1 := 1 TO #ss_NewErrorMessage[#ti_Loop_ItemError_FiFo].Size / #ci_ItemError_BodyLenght DO

	                    #s_UDT_ItemErrorBody := #ss_NewErrorMessage[#ti_Loop_ItemError_FiFo].Body[#ti_Loop_ItemError_FiFo_1];

	                    // Convert message body structure into array of bytes.
	                    #si_BodySerializeStatus := Serialize(SRC_VARIABLE := #s_UDT_ItemErrorBody,
	                                                         DEST_ARRAY => #s_UDT_MessageArray.Bytes,
	                                                         POS := #sdi_SerializePosition);
	                END_FOR;

	                // Mode 'W' - Write FIFO record.
	                "FC_Fifo"(ic_Mode := 'W',
	                          qUDT_Status => #ss_Status.FIFOItemErrorStatus,
	                          qx_Error => #ss_Status.FIFOError,
	                          qx_Warning => #ss_Status.FIFOWarning,
	                          iqv_Data := #s_UDT_MessageArray,
	                          iqUDT_FifoHeader := #iq_UDT_FifoReceiveHeader_Out,
	                          iqv_DataBuffer := #iqs_FifoReceiveData_Out);
	            END_FOR;

	            #si_Counter_ItemError := 0;

	        END_IF;

	    END_REGION

	    REGION 3.2 - Item Status

	        IF #si_Counter_ItemStatus >= 1 THEN

	            #si_NewMessage_Counter := 1;
	            #ss_NewStatusMessage := #ss_NewStatusMessage_Empty;
	            #s_UDT_MessageArray.Bytes := #s_UDT_MessageArray_Empty.Bytes;

	            // Crate new messages
	            FOR #ti_Loop_ItemStatus := 1 TO #si_Counter_ItemStatus DO

	                IF #ss_NewStatusMessage[#si_NewMessage_Counter].Size > #ci_ItemStatus_BodyMaxSize THEN

	                    #si_NewMessage_Counter += 1;

	                END_IF;

	                #ss_NewStatusMessage[#si_NewMessage_Counter].Body[#ti_Loop_ItemStatus] := #sa_Data_ItemStatus[#ti_Loop_ItemStatus];
	                #ss_NewStatusMessage[#si_NewMessage_Counter].Size += 1;

	            END_FOR;


	            FOR #ti_Loop_ItemStatus_FiFo := 1 TO #si_NewMessage_Counter DO

